// TIA Portal V19 export
FUNCTION_BLOCK "A01_HMI_FB"   // FB75, LAD
TITLE = HMI Managment
AUTHOR : Piemme
FAMILY : System
// stored: MemoryReserve 100, SetENOAutomatically false
   VAR
      MB1_Decoder { ExternalAccessible := 'False'; ExternalVisible := 'False'; ExternalWritable := 'False'} : "ButtonsHMIDecoder";
   END_VAR
   VAR CONSTANT
      "1001_HU_AREA01" : Int := 1001;
      "1002_HU_DECOILER" : Int := 1002;
      "1011_DECOILER_IN_LINE_FEED" : Int := 1011;
      "1012_DECOILER_IN_LINE_JAWS" : Int := 1012;
      "1013_DECOILER_IN_LINE_COUPLING" : Int := 1013;
      "1014_DECOILER_IN_LINE_SNUBBER_LIFT" : Int := 1014;
      "1015_DECOILER_IN_LINE_SNUBBER_ROL" : Int := 1015;
      "1016_DECOILER_IN_LINE_BRAKE_OPEN" : Int := 1016;
      "1017_DECOILER_IN_LINE_BRAKE_PARTIAL" : Int := 1017;
      "1021_DECOILER_OUT_LINE_FEED" : Int := 1021;
      "1022_DECOILER_OUT_LINE_JAWS" : Int := 1022;
      "1023_DECOILER_OUT_LINE_COUPLING" : Int := 1023;
      "1024_DECOILER_OUT_LINE_SNUBBER_LIFT" : Int := 1024;
      "1025_DECOILER_OUT_LINE_SNUBBER_ROL" : Int := 1025;
      "1026_DECOILER_OUT_LINE_BRAKE_OPEN" : Int := 1026;
      "1027_DECOILER_OUT_LINE_BRAKE_PARTIAL" : Int := 1027;
      "1031_DECOILER_ROTATION" : Int := 1031;
      "1032_DECOILER_ROTATION_DIR" : Int := 1032;
      "1033_DECOILER_ROTATION_PIVOT" : Int := 1033;
      "1034_DECOILER_TRASLATION_BWD_FWD" : Int := 1034;
      "1035_DECOILER_TRANSLATION_MOVE_TO_POS" : Int := 1035;
      "1041_PEELER_LIFT" : Int := 1041;
      "1042_PEELER_EXTENSION" : Int := 1042;
      "1051_STRAIGHTENER_MOVE" : Int := 1051;
      "1052_STRAIGHTENER_LIFT_ENTRYROLL" : Int := 1052;
      "1053_STRAIGHTENER_LIFT_EXITROLL" : Int := 1053;
      "1054_STRAIGHTENER_COUPLING" : Int := 1054;
      "1061_JB_CUT" : Int := 1061;
      "1062_JB_TORCH_MOVE" : Int := 1062;
      "1063_JB_ENTRYCLAMP" : Int := 1063;
      "1064_JB_EXITCLAMP" : Int := 1064;
      "1065_JB_WELDER" : Int := 1065;
      "1066_JB_WELD_CYCLE" : Int := 1066;
      "1071_JB_PINCHROLL_MOVE" : Int := 1071;
      "1072_JB_PINCHROLL_LIFT" : Int := 1072;
      "1073_JB_PINCHROLL_COUPLING" : Int := 1073;
      "1081_LOOP1" : Int := 1081;
   END_VAR
   VAR_TEMP   // added for the SCL form of the ladder/FBD networks
      _w1 : Bool;
      _w2 : Bool;
   END_VAR
BEGIN

REGION Network 2: <<< MB1 MANUALS OPERATIONS >>>
END_REGION

REGION Network 3 (SCL): Reset Op
   #MB1_Decoder.OpEnabled := FALSE;
   #MB1_Decoder.OpRunning := FALSE;
   #MB1_Decoder.OpDone := FALSE;
END_REGION

REGION Network 4: MB1 Code 1001 - Area 01 HU
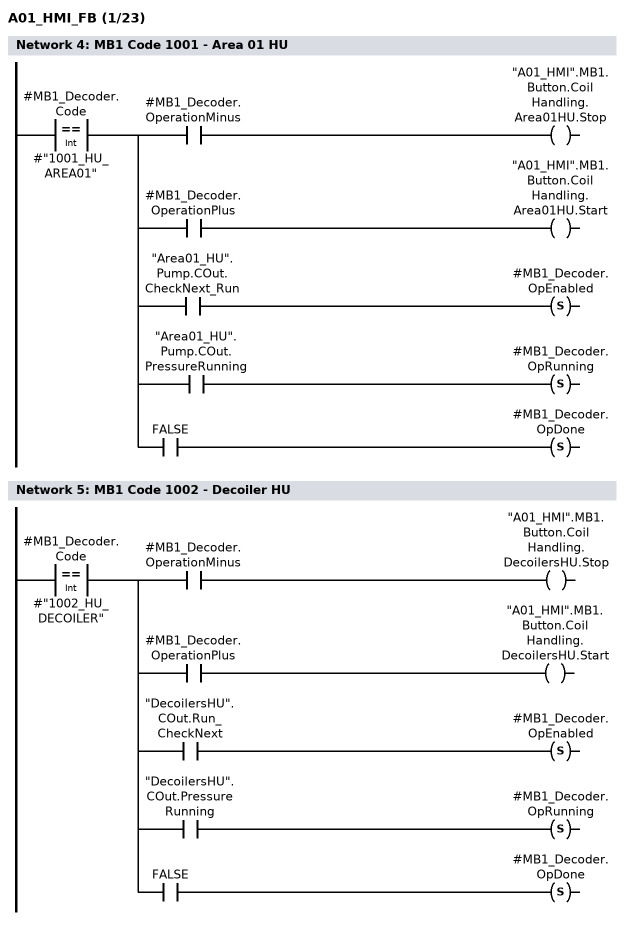
   RUNG wire#powerrail
      { S7_Templates := "SrcType := Int" } EQ_Contact(in1 := #MB1_Decoder.Code, in2 := #"1001_HU_AREA01")
      wire#w1
      Contact( #MB1_Decoder.OperationMinus )
      Coil( "A01_HMI".MB1.Button.CoilHandling.Area01HU.Stop )
   END_RUNG
   RUNG wire#w1
      Contact( #MB1_Decoder.OperationPlus )
      Coil( "A01_HMI".MB1.Button.CoilHandling.Area01HU.Start )
   END_RUNG
   RUNG wire#w1
      Contact( "Area01_HU".Pump.COut.CheckNext_Run )
      S_Coil( #MB1_Decoder.OpEnabled )
   END_RUNG
   RUNG wire#w1
      Contact( "Area01_HU".Pump.COut.PressureRunning )
      S_Coil( #MB1_Decoder.OpRunning )
   END_RUNG
   RUNG wire#w1
      Contact( FALSE )
      S_Coil( #MB1_Decoder.OpDone )
   END_RUNG
   // the same network as SCL:
   #_w1 := #MB1_Decoder.Code = #"1001_HU_AREA01";
   "A01_HMI".MB1.Button.CoilHandling.Area01HU.Stop := #_w1 AND #MB1_Decoder.OperationMinus;
   "A01_HMI".MB1.Button.CoilHandling.Area01HU.Start := #_w1 AND #MB1_Decoder.OperationPlus;
   IF #_w1 AND "Area01_HU".Pump.COut.CheckNext_Run THEN #MB1_Decoder.OpEnabled := TRUE; END_IF;
   IF #_w1 AND "Area01_HU".Pump.COut.PressureRunning THEN #MB1_Decoder.OpRunning := TRUE; END_IF;
   IF #_w1 AND FALSE THEN #MB1_Decoder.OpDone := TRUE; END_IF;
END_REGION

REGION Network 5: MB1 Code 1002 - Decoiler HU
   RUNG wire#powerrail
      { S7_Templates := "SrcType := Int" } EQ_Contact(in1 := #MB1_Decoder.Code, in2 := #"1002_HU_DECOILER")
      wire#w1
      Contact( #MB1_Decoder.OperationMinus )
      Coil( "A01_HMI".MB1.Button.CoilHandling.DecoilersHU.Stop )
   END_RUNG
   RUNG wire#w1
      Contact( #MB1_Decoder.OperationPlus )
      Coil( "A01_HMI".MB1.Button.CoilHandling.DecoilersHU.Start )
   END_RUNG
   RUNG wire#w1
      Contact( "DecoilersHU".COut.Run_CheckNext )
      S_Coil( #MB1_Decoder.OpEnabled )
   END_RUNG
   RUNG wire#w1
      Contact( "DecoilersHU".COut.PressureRunning )
      S_Coil( #MB1_Decoder.OpRunning )
   END_RUNG
   RUNG wire#w1
      Contact( FALSE )
      S_Coil( #MB1_Decoder.OpDone )
   END_RUNG
   // the same network as SCL:
   #_w1 := #MB1_Decoder.Code = #"1002_HU_DECOILER";
   "A01_HMI".MB1.Button.CoilHandling.DecoilersHU.Stop := #_w1 AND #MB1_Decoder.OperationMinus;
   "A01_HMI".MB1.Button.CoilHandling.DecoilersHU.Start := #_w1 AND #MB1_Decoder.OperationPlus;
   IF #_w1 AND "DecoilersHU".COut.Run_CheckNext THEN #MB1_Decoder.OpEnabled := TRUE; END_IF;
   IF #_w1 AND "DecoilersHU".COut.PressureRunning THEN #MB1_Decoder.OpRunning := TRUE; END_IF;
   IF #_w1 AND FALSE THEN #MB1_Decoder.OpDone := TRUE; END_IF;
END_REGION

REGION Network 6: MB1 Code 1011 - Decoiler In Line bkw / fwd
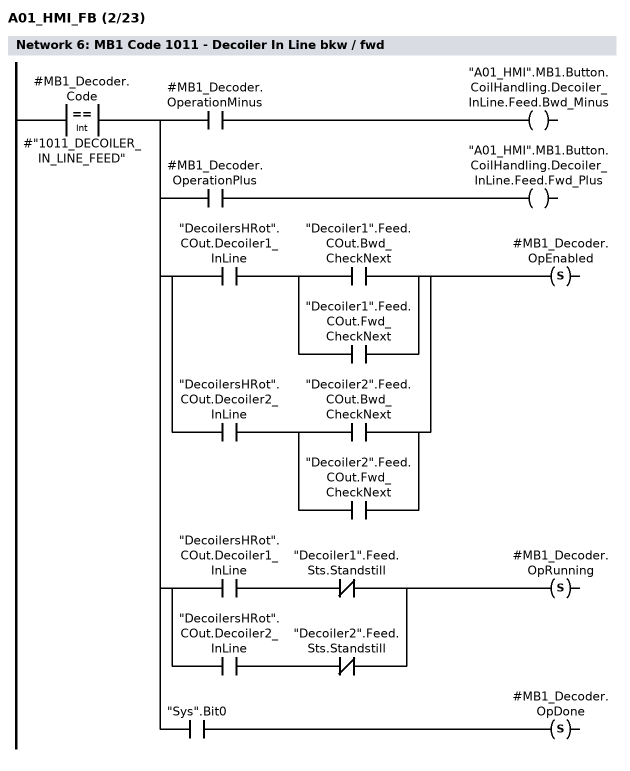
   RUNG wire#powerrail
      { S7_Templates := "SrcType := Int" } EQ_Contact(in1 := #MB1_Decoder.Code, in2 := #"1011_DECOILER_IN_LINE_FEED")
      wire#w1
      Contact( #MB1_Decoder.OperationMinus )
      Coil( "A01_HMI".MB1.Button.CoilHandling.Decoiler_InLine.Feed.Bwd_Minus )
   END_RUNG
   RUNG wire#w1
      Contact( #MB1_Decoder.OperationPlus )
      Coil( "A01_HMI".MB1.Button.CoilHandling.Decoiler_InLine.Feed.Fwd_Plus )
   END_RUNG
   RUNG wire#w1
      Contact( "DecoilersHRot".COut.Decoiler1_InLine )
      wire#w2
      Contact( "Decoiler1".Feed.COut.Bwd_CheckNext )
      wire#w3
      S_Coil( #MB1_Decoder.OpEnabled )
   END_RUNG
   RUNG wire#w2
      Contact( "Decoiler1".Feed.COut.Fwd_CheckNext )
   END_RUNG wire#w3
   RUNG wire#w1
      Contact( "DecoilersHRot".COut.Decoiler2_InLine )
      wire#w4
      Contact( "Decoiler2".Feed.COut.Bwd_CheckNext )
   END_RUNG wire#w3
   RUNG wire#w4
      Contact( "Decoiler2".Feed.COut.Fwd_CheckNext )
   END_RUNG wire#w3
   RUNG wire#w1
      Contact( "DecoilersHRot".COut.Decoiler1_InLine )
      I_Contact( "Decoiler1".Feed.Sts.Standstill )
      wire#w5
      S_Coil( #MB1_Decoder.OpRunning )
   END_RUNG
   RUNG wire#w1
      Contact( "DecoilersHRot".COut.Decoiler2_InLine )
      I_Contact( "Decoiler2".Feed.Sts.Standstill )
   END_RUNG wire#w5
   RUNG wire#w1
      Contact( "Sys".Bit0 )
      S_Coil( #MB1_Decoder.OpDone )
   END_RUNG
   // the same network as SCL:
   #_w1 := #MB1_Decoder.Code = #"1011_DECOILER_IN_LINE_FEED";
   "A01_HMI".MB1.Button.CoilHandling.Decoiler_InLine.Feed.Bwd_Minus := #_w1 AND #MB1_Decoder.OperationMinus;
   "A01_HMI".MB1.Button.CoilHandling.Decoiler_InLine.Feed.Fwd_Plus := #_w1 AND #MB1_Decoder.OperationPlus;
   IF #_w1 AND (("DecoilersHRot".COut.Decoiler1_InLine AND ("Decoiler1".Feed.COut.Bwd_CheckNext OR "Decoiler1".Feed.COut.Fwd_CheckNext)) OR ("DecoilersHRot".COut.Decoiler2_InLine AND ("Decoiler2".Feed.COut.Bwd_CheckNext OR "Decoiler2".Feed.COut.Fwd_CheckNext))) THEN
       #MB1_Decoder.OpEnabled := TRUE;
   END_IF;
   IF #_w1 AND (("DecoilersHRot".COut.Decoiler1_InLine AND NOT "Decoiler1".Feed.Sts.Standstill) OR ("DecoilersHRot".COut.Decoiler2_InLine AND NOT "Decoiler2".Feed.Sts.Standstill)) THEN
       #MB1_Decoder.OpRunning := TRUE;
   END_IF;
   IF #_w1 AND "Sys".Bit0 THEN #MB1_Decoder.OpDone := TRUE; END_IF;
END_REGION

REGION Network 7: MB1 Code 1012 - Decoiler In Line jaws open / close
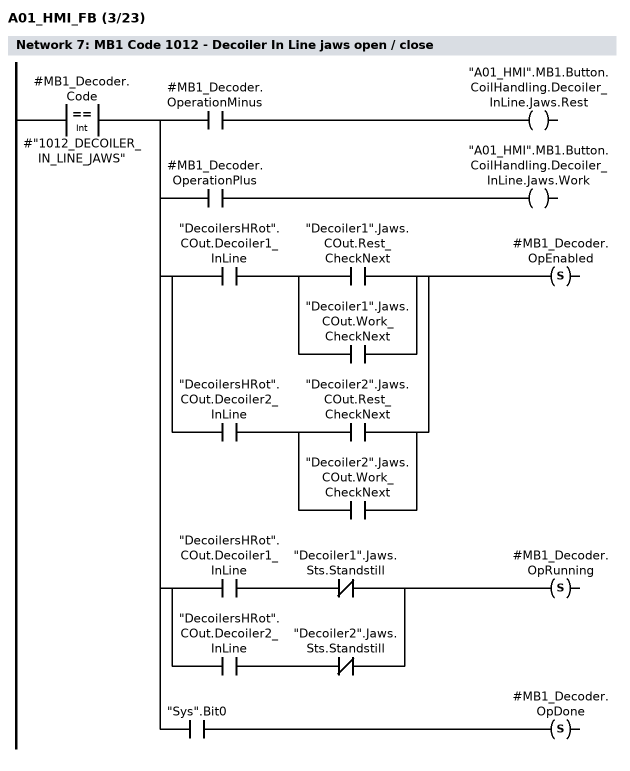
   RUNG wire#powerrail
      { S7_Templates := "SrcType := Int" } EQ_Contact(in1 := #MB1_Decoder.Code, in2 := #"1012_DECOILER_IN_LINE_JAWS")
      wire#w1
      Contact( #MB1_Decoder.OperationMinus )
      Coil( "A01_HMI".MB1.Button.CoilHandling.Decoiler_InLine.Jaws.Rest )
   END_RUNG
   RUNG wire#w1
      Contact( #MB1_Decoder.OperationPlus )
      Coil( "A01_HMI".MB1.Button.CoilHandling.Decoiler_InLine.Jaws.Work )
   END_RUNG
   RUNG wire#w1
      Contact( "DecoilersHRot".COut.Decoiler1_InLine )
      wire#w2
      Contact( "Decoiler1".Jaws.COut.Rest_CheckNext )
      wire#w3
      S_Coil( #MB1_Decoder.OpEnabled )
   END_RUNG
   RUNG wire#w2
      Contact( "Decoiler1".Jaws.COut.Work_CheckNext )
   END_RUNG wire#w3
   RUNG wire#w1
      Contact( "DecoilersHRot".COut.Decoiler2_InLine )
      wire#w4
      Contact( "Decoiler2".Jaws.COut.Rest_CheckNext )
   END_RUNG wire#w3
   RUNG wire#w4
      Contact( "Decoiler2".Jaws.COut.Work_CheckNext )
   END_RUNG wire#w3
   RUNG wire#w1
      Contact( "DecoilersHRot".COut.Decoiler1_InLine )
      I_Contact( "Decoiler1".Jaws.Sts.Standstill )
      wire#w5
      S_Coil( #MB1_Decoder.OpRunning )
   END_RUNG
   RUNG wire#w1
      Contact( "DecoilersHRot".COut.Decoiler2_InLine )
      I_Contact( "Decoiler2".Jaws.Sts.Standstill )
   END_RUNG wire#w5
   RUNG wire#w1
      Contact( "Sys".Bit0 )
      S_Coil( #MB1_Decoder.OpDone )
   END_RUNG
   // the same network as SCL:
   #_w1 := #MB1_Decoder.Code = #"1012_DECOILER_IN_LINE_JAWS";
   "A01_HMI".MB1.Button.CoilHandling.Decoiler_InLine.Jaws.Rest := #_w1 AND #MB1_Decoder.OperationMinus;
   "A01_HMI".MB1.Button.CoilHandling.Decoiler_InLine.Jaws.Work := #_w1 AND #MB1_Decoder.OperationPlus;
   IF #_w1 AND (("DecoilersHRot".COut.Decoiler1_InLine AND ("Decoiler1".Jaws.COut.Rest_CheckNext OR "Decoiler1".Jaws.COut.Work_CheckNext)) OR ("DecoilersHRot".COut.Decoiler2_InLine AND ("Decoiler2".Jaws.COut.Rest_CheckNext OR "Decoiler2".Jaws.COut.Work_CheckNext))) THEN
       #MB1_Decoder.OpEnabled := TRUE;
   END_IF;
   IF #_w1 AND (("DecoilersHRot".COut.Decoiler1_InLine AND NOT "Decoiler1".Jaws.Sts.Standstill) OR ("DecoilersHRot".COut.Decoiler2_InLine AND NOT "Decoiler2".Jaws.Sts.Standstill)) THEN
       #MB1_Decoder.OpRunning := TRUE;
   END_IF;
   IF #_w1 AND "Sys".Bit0 THEN #MB1_Decoder.OpDone := TRUE; END_IF;
END_REGION

REGION Network 8: MB1 Code 1013 - Decoiler In Line motor coupling rest / work
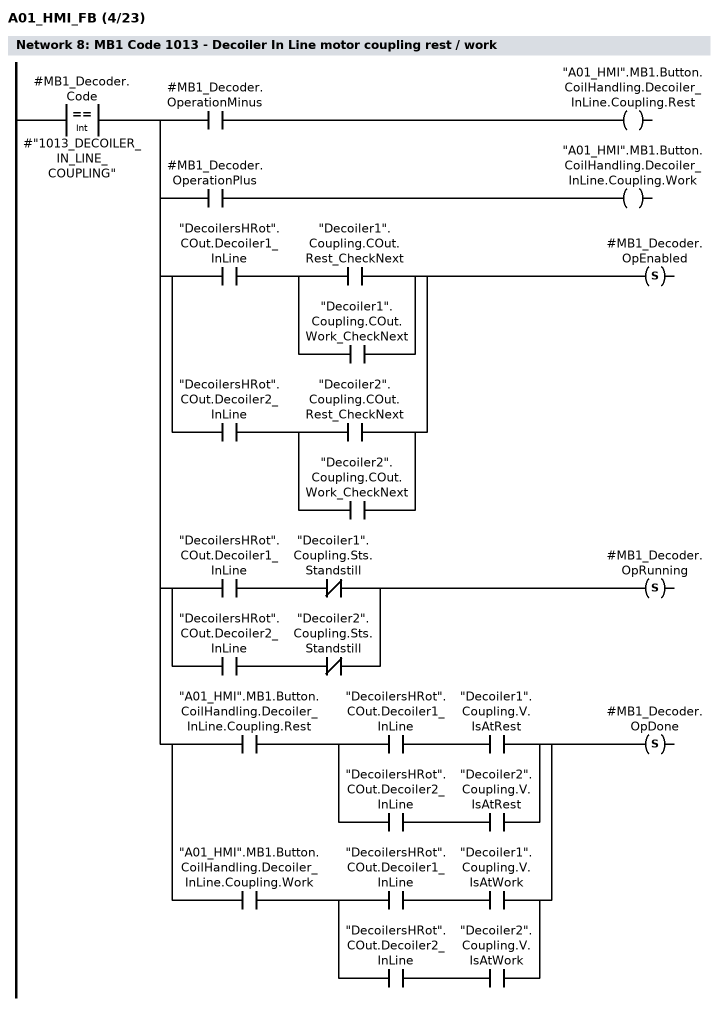
   RUNG wire#powerrail
      { S7_Templates := "SrcType := Int" } EQ_Contact(in1 := #MB1_Decoder.Code, in2 := #"1013_DECOILER_IN_LINE_COUPLING")
      wire#w1
      Contact( #MB1_Decoder.OperationMinus )
      Coil( "A01_HMI".MB1.Button.CoilHandling.Decoiler_InLine.Coupling.Rest )
   END_RUNG
   RUNG wire#w1
      Contact( #MB1_Decoder.OperationPlus )
      Coil( "A01_HMI".MB1.Button.CoilHandling.Decoiler_InLine.Coupling.Work )
   END_RUNG
   RUNG wire#w1
      Contact( "DecoilersHRot".COut.Decoiler1_InLine )
      wire#w2
      Contact( "Decoiler1".Coupling.COut.Rest_CheckNext )
      wire#w3
      S_Coil( #MB1_Decoder.OpEnabled )
   END_RUNG
   RUNG wire#w2
      Contact( "Decoiler1".Coupling.COut.Work_CheckNext )
   END_RUNG wire#w3
   RUNG wire#w1
      Contact( "DecoilersHRot".COut.Decoiler2_InLine )
      wire#w4
      Contact( "Decoiler2".Coupling.COut.Rest_CheckNext )
   END_RUNG wire#w3
   RUNG wire#w4
      Contact( "Decoiler2".Coupling.COut.Work_CheckNext )
   END_RUNG wire#w3
   RUNG wire#w1
      Contact( "DecoilersHRot".COut.Decoiler1_InLine )
      I_Contact( "Decoiler1".Coupling.Sts.Standstill )
      wire#w5
      S_Coil( #MB1_Decoder.OpRunning )
   END_RUNG
   RUNG wire#w1
      Contact( "DecoilersHRot".COut.Decoiler2_InLine )
      I_Contact( "Decoiler2".Coupling.Sts.Standstill )
   END_RUNG wire#w5
   RUNG wire#w1
      Contact( "A01_HMI".MB1.Button.CoilHandling.Decoiler_InLine.Coupling.Rest )
      wire#w6
      Contact( "DecoilersHRot".COut.Decoiler1_InLine )
      Contact( "Decoiler1".Coupling.V.IsAtRest )
      wire#w7
      S_Coil( #MB1_Decoder.OpDone )
   END_RUNG
   RUNG wire#w6
      Contact( "DecoilersHRot".COut.Decoiler2_InLine )
      Contact( "Decoiler2".Coupling.V.IsAtRest )
   END_RUNG wire#w7
   RUNG wire#w1
      Contact( "A01_HMI".MB1.Button.CoilHandling.Decoiler_InLine.Coupling.Work )
      wire#w8
      Contact( "DecoilersHRot".COut.Decoiler1_InLine )
      Contact( "Decoiler1".Coupling.V.IsAtWork )
   END_RUNG wire#w7
   RUNG wire#w8
      Contact( "DecoilersHRot".COut.Decoiler2_InLine )
      Contact( "Decoiler2".Coupling.V.IsAtWork )
   END_RUNG wire#w7
   // the same network as SCL:
   #_w1 := #MB1_Decoder.Code = #"1013_DECOILER_IN_LINE_COUPLING";
   "A01_HMI".MB1.Button.CoilHandling.Decoiler_InLine.Coupling.Rest := #_w1 AND #MB1_Decoder.OperationMinus;
   "A01_HMI".MB1.Button.CoilHandling.Decoiler_InLine.Coupling.Work := #_w1 AND #MB1_Decoder.OperationPlus;
   IF #_w1 AND (("DecoilersHRot".COut.Decoiler1_InLine AND ("Decoiler1".Coupling.COut.Rest_CheckNext OR "Decoiler1".Coupling.COut.Work_CheckNext)) OR ("DecoilersHRot".COut.Decoiler2_InLine AND ("Decoiler2".Coupling.COut.Rest_CheckNext OR "Decoiler2".Coupling.COut.Work_CheckNext))) THEN
       #MB1_Decoder.OpEnabled := TRUE;
   END_IF;
   IF #_w1 AND (("DecoilersHRot".COut.Decoiler1_InLine AND NOT "Decoiler1".Coupling.Sts.Standstill) OR ("DecoilersHRot".COut.Decoiler2_InLine AND NOT "Decoiler2".Coupling.Sts.Standstill)) THEN
       #MB1_Decoder.OpRunning := TRUE;
   END_IF;
   IF #_w1 AND (("A01_HMI".MB1.Button.CoilHandling.Decoiler_InLine.Coupling.Rest AND (("DecoilersHRot".COut.Decoiler1_InLine AND "Decoiler1".Coupling.V.IsAtRest) OR ("DecoilersHRot".COut.Decoiler2_InLine AND "Decoiler2".Coupling.V.IsAtRest))) OR ("A01_HMI".MB1.Button.CoilHandling.Decoiler_InLine.Coupling.Work AND (("DecoilersHRot".COut.Decoiler1_InLine AND "Decoiler1".Coupling.V.IsAtWork) OR ("DecoilersHRot".COut.Decoiler2_InLine AND "Decoiler2".Coupling.V.IsAtWork)))) THEN
       #MB1_Decoder.OpDone := TRUE;
   END_IF;
END_REGION

REGION Network 9: MB1 Code 1014 - Decoiler In Line snubber lift up / down
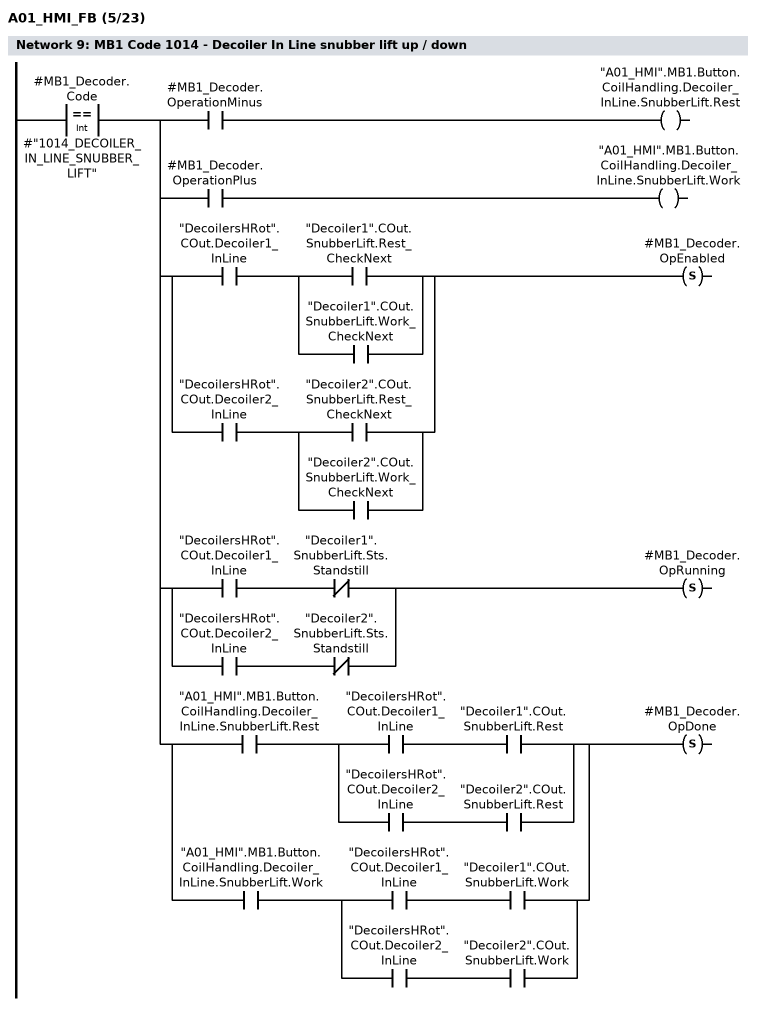
   RUNG wire#powerrail
      { S7_Templates := "SrcType := Int" } EQ_Contact(in1 := #MB1_Decoder.Code, in2 := #"1014_DECOILER_IN_LINE_SNUBBER_LIFT")
      wire#w1
      Contact( #MB1_Decoder.OperationMinus )
      Coil( "A01_HMI".MB1.Button.CoilHandling.Decoiler_InLine.SnubberLift.Rest )
   END_RUNG
   RUNG wire#w1
      Contact( #MB1_Decoder.OperationPlus )
      Coil( "A01_HMI".MB1.Button.CoilHandling.Decoiler_InLine.SnubberLift.Work )
   END_RUNG
   RUNG wire#w1
      Contact( "DecoilersHRot".COut.Decoiler1_InLine )
      wire#w2
      Contact( "Decoiler1".COut.SnubberLift.Rest_CheckNext )
      wire#w3
      S_Coil( #MB1_Decoder.OpEnabled )
   END_RUNG
   RUNG wire#w2
      Contact( "Decoiler1".COut.SnubberLift.Work_CheckNext )
   END_RUNG wire#w3
   RUNG wire#w1
      Contact( "DecoilersHRot".COut.Decoiler2_InLine )
      wire#w4
      Contact( "Decoiler2".COut.SnubberLift.Rest_CheckNext )
   END_RUNG wire#w3
   RUNG wire#w4
      Contact( "Decoiler2".COut.SnubberLift.Work_CheckNext )
   END_RUNG wire#w3
   RUNG wire#w1
      Contact( "DecoilersHRot".COut.Decoiler1_InLine )
      I_Contact( "Decoiler1".SnubberLift.Sts.Standstill )
      wire#w5
      S_Coil( #MB1_Decoder.OpRunning )
   END_RUNG
   RUNG wire#w1
      Contact( "DecoilersHRot".COut.Decoiler2_InLine )
      I_Contact( "Decoiler2".SnubberLift.Sts.Standstill )
   END_RUNG wire#w5
   RUNG wire#w1
      Contact( "A01_HMI".MB1.Button.CoilHandling.Decoiler_InLine.SnubberLift.Rest )
      wire#w6
      Contact( "DecoilersHRot".COut.Decoiler1_InLine )
      Contact( "Decoiler1".COut.SnubberLift.Rest )
      wire#w7
      S_Coil( #MB1_Decoder.OpDone )
   END_RUNG
   RUNG wire#w6
      Contact( "DecoilersHRot".COut.Decoiler2_InLine )
      Contact( "Decoiler2".COut.SnubberLift.Rest )
   END_RUNG wire#w7
   RUNG wire#w1
      Contact( "A01_HMI".MB1.Button.CoilHandling.Decoiler_InLine.SnubberLift.Work )
      wire#w8
      Contact( "DecoilersHRot".COut.Decoiler1_InLine )
      Contact( "Decoiler1".COut.SnubberLift.Work )
   END_RUNG wire#w7
   RUNG wire#w8
      Contact( "DecoilersHRot".COut.Decoiler2_InLine )
      Contact( "Decoiler2".COut.SnubberLift.Work )
   END_RUNG wire#w7
   // the same network as SCL:
   #_w1 := #MB1_Decoder.Code = #"1014_DECOILER_IN_LINE_SNUBBER_LIFT";
   "A01_HMI".MB1.Button.CoilHandling.Decoiler_InLine.SnubberLift.Rest := #_w1 AND #MB1_Decoder.OperationMinus;
   "A01_HMI".MB1.Button.CoilHandling.Decoiler_InLine.SnubberLift.Work := #_w1 AND #MB1_Decoder.OperationPlus;
   IF #_w1 AND (("DecoilersHRot".COut.Decoiler1_InLine AND ("Decoiler1".COut.SnubberLift.Rest_CheckNext OR "Decoiler1".COut.SnubberLift.Work_CheckNext)) OR ("DecoilersHRot".COut.Decoiler2_InLine AND ("Decoiler2".COut.SnubberLift.Rest_CheckNext OR "Decoiler2".COut.SnubberLift.Work_CheckNext))) THEN
       #MB1_Decoder.OpEnabled := TRUE;
   END_IF;
   IF #_w1 AND (("DecoilersHRot".COut.Decoiler1_InLine AND NOT "Decoiler1".SnubberLift.Sts.Standstill) OR ("DecoilersHRot".COut.Decoiler2_InLine AND NOT "Decoiler2".SnubberLift.Sts.Standstill)) THEN
       #MB1_Decoder.OpRunning := TRUE;
   END_IF;
   IF #_w1 AND (("A01_HMI".MB1.Button.CoilHandling.Decoiler_InLine.SnubberLift.Rest AND (("DecoilersHRot".COut.Decoiler1_InLine AND "Decoiler1".COut.SnubberLift.Rest) OR ("DecoilersHRot".COut.Decoiler2_InLine AND "Decoiler2".COut.SnubberLift.Rest))) OR ("A01_HMI".MB1.Button.CoilHandling.Decoiler_InLine.SnubberLift.Work AND (("DecoilersHRot".COut.Decoiler1_InLine AND "Decoiler1".COut.SnubberLift.Work) OR ("DecoilersHRot".COut.Decoiler2_InLine AND "Decoiler2".COut.SnubberLift.Work)))) THEN
       #MB1_Decoder.OpDone := TRUE;
   END_IF;
END_REGION

REGION Network 10: MB1 Code 1015 - Decoiler In Line nubber roll bkw / fwd
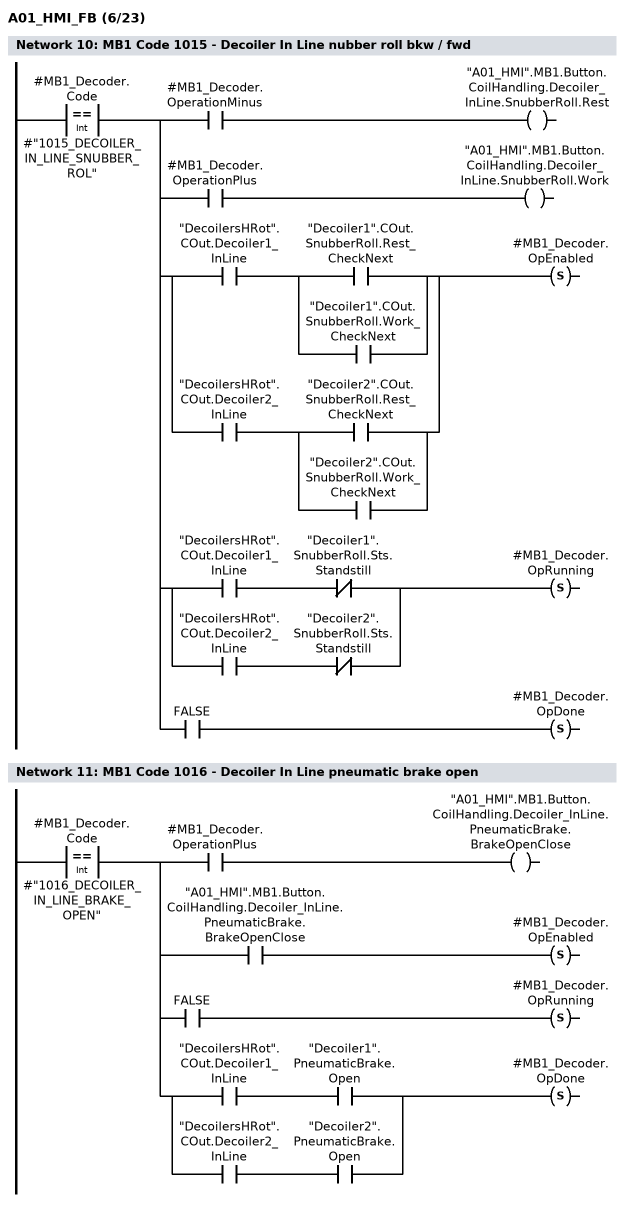
   RUNG wire#powerrail
      { S7_Templates := "SrcType := Int" } EQ_Contact(in1 := #MB1_Decoder.Code, in2 := #"1015_DECOILER_IN_LINE_SNUBBER_ROL")
      wire#w1
      Contact( #MB1_Decoder.OperationMinus )
      Coil( "A01_HMI".MB1.Button.CoilHandling.Decoiler_InLine.SnubberRoll.Rest )
   END_RUNG
   RUNG wire#w1
      Contact( #MB1_Decoder.OperationPlus )
      Coil( "A01_HMI".MB1.Button.CoilHandling.Decoiler_InLine.SnubberRoll.Work )
   END_RUNG
   RUNG wire#w1
      Contact( "DecoilersHRot".COut.Decoiler1_InLine )
      wire#w2
      Contact( "Decoiler1".COut.SnubberRoll.Rest_CheckNext )
      wire#w3
      S_Coil( #MB1_Decoder.OpEnabled )
   END_RUNG
   RUNG wire#w2
      Contact( "Decoiler1".COut.SnubberRoll.Work_CheckNext )
   END_RUNG wire#w3
   RUNG wire#w1
      Contact( "DecoilersHRot".COut.Decoiler2_InLine )
      wire#w4
      Contact( "Decoiler2".COut.SnubberRoll.Rest_CheckNext )
   END_RUNG wire#w3
   RUNG wire#w4
      Contact( "Decoiler2".COut.SnubberRoll.Work_CheckNext )
   END_RUNG wire#w3
   RUNG wire#w1
      Contact( "DecoilersHRot".COut.Decoiler1_InLine )
      I_Contact( "Decoiler1".SnubberRoll.Sts.Standstill )
      wire#w5
      S_Coil( #MB1_Decoder.OpRunning )
   END_RUNG
   RUNG wire#w1
      Contact( "DecoilersHRot".COut.Decoiler2_InLine )
      I_Contact( "Decoiler2".SnubberRoll.Sts.Standstill )
   END_RUNG wire#w5
   RUNG wire#w1
      Contact( FALSE )
      S_Coil( #MB1_Decoder.OpDone )
   END_RUNG
   // the same network as SCL:
   #_w1 := #MB1_Decoder.Code = #"1015_DECOILER_IN_LINE_SNUBBER_ROL";
   "A01_HMI".MB1.Button.CoilHandling.Decoiler_InLine.SnubberRoll.Rest := #_w1 AND #MB1_Decoder.OperationMinus;
   "A01_HMI".MB1.Button.CoilHandling.Decoiler_InLine.SnubberRoll.Work := #_w1 AND #MB1_Decoder.OperationPlus;
   IF #_w1 AND (("DecoilersHRot".COut.Decoiler1_InLine AND ("Decoiler1".COut.SnubberRoll.Rest_CheckNext OR "Decoiler1".COut.SnubberRoll.Work_CheckNext)) OR ("DecoilersHRot".COut.Decoiler2_InLine AND ("Decoiler2".COut.SnubberRoll.Rest_CheckNext OR "Decoiler2".COut.SnubberRoll.Work_CheckNext))) THEN
       #MB1_Decoder.OpEnabled := TRUE;
   END_IF;
   IF #_w1 AND (("DecoilersHRot".COut.Decoiler1_InLine AND NOT "Decoiler1".SnubberRoll.Sts.Standstill) OR ("DecoilersHRot".COut.Decoiler2_InLine AND NOT "Decoiler2".SnubberRoll.Sts.Standstill)) THEN
       #MB1_Decoder.OpRunning := TRUE;
   END_IF;
   IF #_w1 AND FALSE THEN #MB1_Decoder.OpDone := TRUE; END_IF;
END_REGION

REGION Network 11: MB1 Code 1016 - Decoiler In Line pneumatic brake open
   RUNG wire#powerrail
      { S7_Templates := "SrcType := Int" } EQ_Contact(in1 := #MB1_Decoder.Code, in2 := #"1016_DECOILER_IN_LINE_BRAKE_OPEN")
      wire#w1
      Contact( #MB1_Decoder.OperationPlus )
      Coil( "A01_HMI".MB1.Button.CoilHandling.Decoiler_InLine.PneumaticBrake.BrakeOpenClose )
   END_RUNG
   RUNG wire#w1
      Contact( "A01_HMI".MB1.Button.CoilHandling.Decoiler_InLine.PneumaticBrake.BrakeOpenClose )
      S_Coil( #MB1_Decoder.OpEnabled )
   END_RUNG
   RUNG wire#w1
      Contact( FALSE )
      S_Coil( #MB1_Decoder.OpRunning )
   END_RUNG
   RUNG wire#w1
      Contact( "DecoilersHRot".COut.Decoiler1_InLine )
      Contact( "Decoiler1".PneumaticBrake.Open )
      wire#w2
      S_Coil( #MB1_Decoder.OpDone )
   END_RUNG
   RUNG wire#w1
      Contact( "DecoilersHRot".COut.Decoiler2_InLine )
      Contact( "Decoiler2".PneumaticBrake.Open )
   END_RUNG wire#w2
   // the same network as SCL:
   #_w1 := #MB1_Decoder.Code = #"1016_DECOILER_IN_LINE_BRAKE_OPEN";
   "A01_HMI".MB1.Button.CoilHandling.Decoiler_InLine.PneumaticBrake.BrakeOpenClose := #_w1 AND #MB1_Decoder.OperationPlus;
   IF #_w1 AND "A01_HMI".MB1.Button.CoilHandling.Decoiler_InLine.PneumaticBrake.BrakeOpenClose THEN
       #MB1_Decoder.OpEnabled := TRUE;
   END_IF;
   IF #_w1 AND FALSE THEN #MB1_Decoder.OpRunning := TRUE; END_IF;
   IF #_w1 AND (("DecoilersHRot".COut.Decoiler1_InLine AND "Decoiler1".PneumaticBrake.Open) OR ("DecoilersHRot".COut.Decoiler2_InLine AND "Decoiler2".PneumaticBrake.Open)) THEN
       #MB1_Decoder.OpDone := TRUE;
   END_IF;
END_REGION

REGION Network 12: MB1 Code 1017 - Decoiler In Line pneumatic brake partial
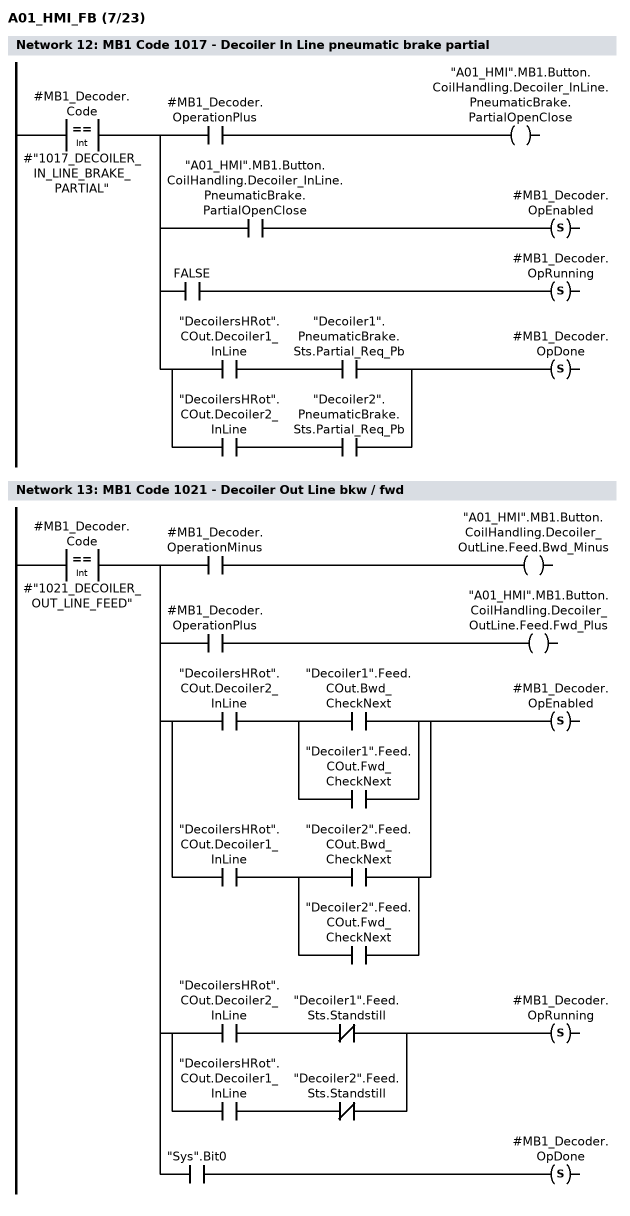
   RUNG wire#powerrail
      { S7_Templates := "SrcType := Int" } EQ_Contact(in1 := #MB1_Decoder.Code, in2 := #"1017_DECOILER_IN_LINE_BRAKE_PARTIAL")
      wire#w1
      Contact( #MB1_Decoder.OperationPlus )
      Coil( "A01_HMI".MB1.Button.CoilHandling.Decoiler_InLine.PneumaticBrake.PartialOpenClose )
   END_RUNG
   RUNG wire#w1
      Contact( "A01_HMI".MB1.Button.CoilHandling.Decoiler_InLine.PneumaticBrake.PartialOpenClose )
      S_Coil( #MB1_Decoder.OpEnabled )
   END_RUNG
   RUNG wire#w1
      Contact( FALSE )
      S_Coil( #MB1_Decoder.OpRunning )
   END_RUNG
   RUNG wire#w1
      Contact( "DecoilersHRot".COut.Decoiler1_InLine )
      Contact( "Decoiler1".PneumaticBrake.Sts.Partial_Req_Pb )
      wire#w2
      S_Coil( #MB1_Decoder.OpDone )
   END_RUNG
   RUNG wire#w1
      Contact( "DecoilersHRot".COut.Decoiler2_InLine )
      Contact( "Decoiler2".PneumaticBrake.Sts.Partial_Req_Pb )
   END_RUNG wire#w2
   // the same network as SCL:
   #_w1 := #MB1_Decoder.Code = #"1017_DECOILER_IN_LINE_BRAKE_PARTIAL";
   "A01_HMI".MB1.Button.CoilHandling.Decoiler_InLine.PneumaticBrake.PartialOpenClose := #_w1 AND #MB1_Decoder.OperationPlus;
   IF #_w1 AND "A01_HMI".MB1.Button.CoilHandling.Decoiler_InLine.PneumaticBrake.PartialOpenClose THEN
       #MB1_Decoder.OpEnabled := TRUE;
   END_IF;
   IF #_w1 AND FALSE THEN #MB1_Decoder.OpRunning := TRUE; END_IF;
   IF #_w1 AND (("DecoilersHRot".COut.Decoiler1_InLine AND "Decoiler1".PneumaticBrake.Sts.Partial_Req_Pb) OR ("DecoilersHRot".COut.Decoiler2_InLine AND "Decoiler2".PneumaticBrake.Sts.Partial_Req_Pb)) THEN
       #MB1_Decoder.OpDone := TRUE;
   END_IF;
END_REGION

REGION Network 13: MB1 Code 1021 - Decoiler Out Line bkw / fwd
   RUNG wire#powerrail
      { S7_Templates := "SrcType := Int" } EQ_Contact(in1 := #MB1_Decoder.Code, in2 := #"1021_DECOILER_OUT_LINE_FEED")
      wire#w1
      Contact( #MB1_Decoder.OperationMinus )
      Coil( "A01_HMI".MB1.Button.CoilHandling.Decoiler_OutLine.Feed.Bwd_Minus )
   END_RUNG
   RUNG wire#w1
      Contact( #MB1_Decoder.OperationPlus )
      Coil( "A01_HMI".MB1.Button.CoilHandling.Decoiler_OutLine.Feed.Fwd_Plus )
   END_RUNG
   RUNG wire#w1
      Contact( "DecoilersHRot".COut.Decoiler2_InLine )
      wire#w2
      Contact( "Decoiler1".Feed.COut.Bwd_CheckNext )
      wire#w3
      S_Coil( #MB1_Decoder.OpEnabled )
   END_RUNG
   RUNG wire#w2
      Contact( "Decoiler1".Feed.COut.Fwd_CheckNext )
   END_RUNG wire#w3
   RUNG wire#w1
      Contact( "DecoilersHRot".COut.Decoiler1_InLine )
      wire#w4
      Contact( "Decoiler2".Feed.COut.Bwd_CheckNext )
   END_RUNG wire#w3
   RUNG wire#w4
      Contact( "Decoiler2".Feed.COut.Fwd_CheckNext )
   END_RUNG wire#w3
   RUNG wire#w1
      Contact( "DecoilersHRot".COut.Decoiler2_InLine )
      I_Contact( "Decoiler1".Feed.Sts.Standstill )
      wire#w5
      S_Coil( #MB1_Decoder.OpRunning )
   END_RUNG
   RUNG wire#w1
      Contact( "DecoilersHRot".COut.Decoiler1_InLine )
      I_Contact( "Decoiler2".Feed.Sts.Standstill )
   END_RUNG wire#w5
   RUNG wire#w1
      Contact( "Sys".Bit0 )
      S_Coil( #MB1_Decoder.OpDone )
   END_RUNG
   // the same network as SCL:
   #_w1 := #MB1_Decoder.Code = #"1021_DECOILER_OUT_LINE_FEED";
   "A01_HMI".MB1.Button.CoilHandling.Decoiler_OutLine.Feed.Bwd_Minus := #_w1 AND #MB1_Decoder.OperationMinus;
   "A01_HMI".MB1.Button.CoilHandling.Decoiler_OutLine.Feed.Fwd_Plus := #_w1 AND #MB1_Decoder.OperationPlus;
   IF #_w1 AND (("DecoilersHRot".COut.Decoiler2_InLine AND ("Decoiler1".Feed.COut.Bwd_CheckNext OR "Decoiler1".Feed.COut.Fwd_CheckNext)) OR ("DecoilersHRot".COut.Decoiler1_InLine AND ("Decoiler2".Feed.COut.Bwd_CheckNext OR "Decoiler2".Feed.COut.Fwd_CheckNext))) THEN
       #MB1_Decoder.OpEnabled := TRUE;
   END_IF;
   IF #_w1 AND (("DecoilersHRot".COut.Decoiler2_InLine AND NOT "Decoiler1".Feed.Sts.Standstill) OR ("DecoilersHRot".COut.Decoiler1_InLine AND NOT "Decoiler2".Feed.Sts.Standstill)) THEN
       #MB1_Decoder.OpRunning := TRUE;
   END_IF;
   IF #_w1 AND "Sys".Bit0 THEN #MB1_Decoder.OpDone := TRUE; END_IF;
END_REGION

REGION Network 14: MB1 Code 1022 - Decoiler Out Line jaws open / close
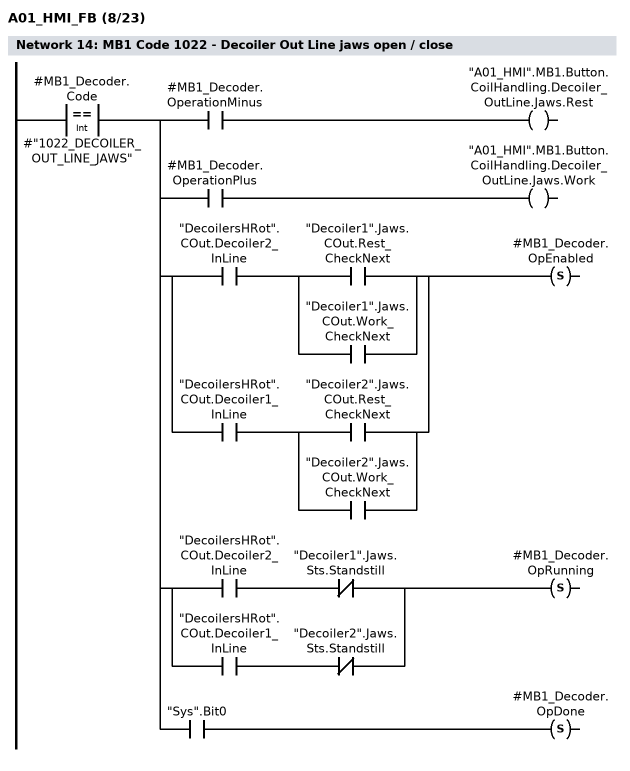
   RUNG wire#powerrail
      { S7_Templates := "SrcType := Int" } EQ_Contact(in1 := #MB1_Decoder.Code, in2 := #"1022_DECOILER_OUT_LINE_JAWS")
      wire#w1
      Contact( #MB1_Decoder.OperationMinus )
      Coil( "A01_HMI".MB1.Button.CoilHandling.Decoiler_OutLine.Jaws.Rest )
   END_RUNG
   RUNG wire#w1
      Contact( #MB1_Decoder.OperationPlus )
      Coil( "A01_HMI".MB1.Button.CoilHandling.Decoiler_OutLine.Jaws.Work )
   END_RUNG
   RUNG wire#w1
      Contact( "DecoilersHRot".COut.Decoiler2_InLine )
      wire#w2
      Contact( "Decoiler1".Jaws.COut.Rest_CheckNext )
      wire#w3
      S_Coil( #MB1_Decoder.OpEnabled )
   END_RUNG
   RUNG wire#w2
      Contact( "Decoiler1".Jaws.COut.Work_CheckNext )
   END_RUNG wire#w3
   RUNG wire#w1
      Contact( "DecoilersHRot".COut.Decoiler1_InLine )
      wire#w4
      Contact( "Decoiler2".Jaws.COut.Rest_CheckNext )
   END_RUNG wire#w3
   RUNG wire#w4
      Contact( "Decoiler2".Jaws.COut.Work_CheckNext )
   END_RUNG wire#w3
   RUNG wire#w1
      Contact( "DecoilersHRot".COut.Decoiler2_InLine )
      I_Contact( "Decoiler1".Jaws.Sts.Standstill )
      wire#w5
      S_Coil( #MB1_Decoder.OpRunning )
   END_RUNG
   RUNG wire#w1
      Contact( "DecoilersHRot".COut.Decoiler1_InLine )
      I_Contact( "Decoiler2".Jaws.Sts.Standstill )
   END_RUNG wire#w5
   RUNG wire#w1
      Contact( "Sys".Bit0 )
      S_Coil( #MB1_Decoder.OpDone )
   END_RUNG
   // the same network as SCL:
   #_w1 := #MB1_Decoder.Code = #"1022_DECOILER_OUT_LINE_JAWS";
   "A01_HMI".MB1.Button.CoilHandling.Decoiler_OutLine.Jaws.Rest := #_w1 AND #MB1_Decoder.OperationMinus;
   "A01_HMI".MB1.Button.CoilHandling.Decoiler_OutLine.Jaws.Work := #_w1 AND #MB1_Decoder.OperationPlus;
   IF #_w1 AND (("DecoilersHRot".COut.Decoiler2_InLine AND ("Decoiler1".Jaws.COut.Rest_CheckNext OR "Decoiler1".Jaws.COut.Work_CheckNext)) OR ("DecoilersHRot".COut.Decoiler1_InLine AND ("Decoiler2".Jaws.COut.Rest_CheckNext OR "Decoiler2".Jaws.COut.Work_CheckNext))) THEN
       #MB1_Decoder.OpEnabled := TRUE;
   END_IF;
   IF #_w1 AND (("DecoilersHRot".COut.Decoiler2_InLine AND NOT "Decoiler1".Jaws.Sts.Standstill) OR ("DecoilersHRot".COut.Decoiler1_InLine AND NOT "Decoiler2".Jaws.Sts.Standstill)) THEN
       #MB1_Decoder.OpRunning := TRUE;
   END_IF;
   IF #_w1 AND "Sys".Bit0 THEN #MB1_Decoder.OpDone := TRUE; END_IF;
END_REGION

REGION Network 15: MB1 Code 1023 - Decoiler Out Line motor coupling rest / work
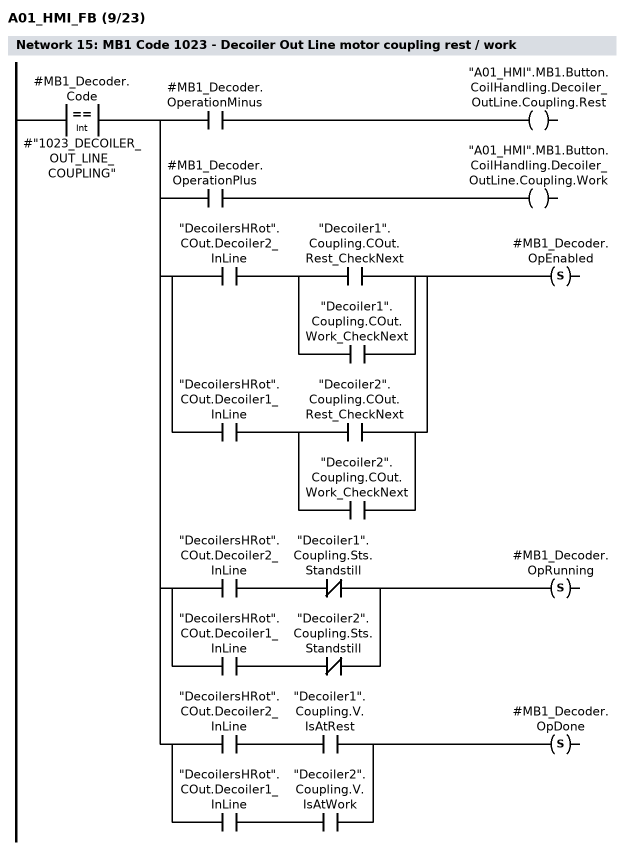
   RUNG wire#powerrail
      { S7_Templates := "SrcType := Int" } EQ_Contact(in1 := #MB1_Decoder.Code, in2 := #"1023_DECOILER_OUT_LINE_COUPLING")
      wire#w1
      Contact( #MB1_Decoder.OperationMinus )
      Coil( "A01_HMI".MB1.Button.CoilHandling.Decoiler_OutLine.Coupling.Rest )
   END_RUNG
   RUNG wire#w1
      Contact( #MB1_Decoder.OperationPlus )
      Coil( "A01_HMI".MB1.Button.CoilHandling.Decoiler_OutLine.Coupling.Work )
   END_RUNG
   RUNG wire#w1
      Contact( "DecoilersHRot".COut.Decoiler2_InLine )
      wire#w2
      Contact( "Decoiler1".Coupling.COut.Rest_CheckNext )
      wire#w3
      S_Coil( #MB1_Decoder.OpEnabled )
   END_RUNG
   RUNG wire#w2
      Contact( "Decoiler1".Coupling.COut.Work_CheckNext )
   END_RUNG wire#w3
   RUNG wire#w1
      Contact( "DecoilersHRot".COut.Decoiler1_InLine )
      wire#w4
      Contact( "Decoiler2".Coupling.COut.Rest_CheckNext )
   END_RUNG wire#w3
   RUNG wire#w4
      Contact( "Decoiler2".Coupling.COut.Work_CheckNext )
   END_RUNG wire#w3
   RUNG wire#w1
      Contact( "DecoilersHRot".COut.Decoiler2_InLine )
      I_Contact( "Decoiler1".Coupling.Sts.Standstill )
      wire#w5
      S_Coil( #MB1_Decoder.OpRunning )
   END_RUNG
   RUNG wire#w1
      Contact( "DecoilersHRot".COut.Decoiler1_InLine )
      I_Contact( "Decoiler2".Coupling.Sts.Standstill )
   END_RUNG wire#w5
   RUNG wire#w1
      Contact( "DecoilersHRot".COut.Decoiler2_InLine )
      Contact( "Decoiler1".Coupling.V.IsAtRest )
      wire#w6
      S_Coil( #MB1_Decoder.OpDone )
   END_RUNG
   RUNG wire#w1
      Contact( "DecoilersHRot".COut.Decoiler1_InLine )
      Contact( "Decoiler2".Coupling.V.IsAtWork )
   END_RUNG wire#w6
   // the same network as SCL:
   #_w1 := #MB1_Decoder.Code = #"1023_DECOILER_OUT_LINE_COUPLING";
   "A01_HMI".MB1.Button.CoilHandling.Decoiler_OutLine.Coupling.Rest := #_w1 AND #MB1_Decoder.OperationMinus;
   "A01_HMI".MB1.Button.CoilHandling.Decoiler_OutLine.Coupling.Work := #_w1 AND #MB1_Decoder.OperationPlus;
   IF #_w1 AND (("DecoilersHRot".COut.Decoiler2_InLine AND ("Decoiler1".Coupling.COut.Rest_CheckNext OR "Decoiler1".Coupling.COut.Work_CheckNext)) OR ("DecoilersHRot".COut.Decoiler1_InLine AND ("Decoiler2".Coupling.COut.Rest_CheckNext OR "Decoiler2".Coupling.COut.Work_CheckNext))) THEN
       #MB1_Decoder.OpEnabled := TRUE;
   END_IF;
   IF #_w1 AND (("DecoilersHRot".COut.Decoiler2_InLine AND NOT "Decoiler1".Coupling.Sts.Standstill) OR ("DecoilersHRot".COut.Decoiler1_InLine AND NOT "Decoiler2".Coupling.Sts.Standstill)) THEN
       #MB1_Decoder.OpRunning := TRUE;
   END_IF;
   IF #_w1 AND (("DecoilersHRot".COut.Decoiler2_InLine AND "Decoiler1".Coupling.V.IsAtRest) OR ("DecoilersHRot".COut.Decoiler1_InLine AND "Decoiler2".Coupling.V.IsAtWork)) THEN
       #MB1_Decoder.OpDone := TRUE;
   END_IF;
END_REGION

REGION Network 16: MB1 Code 1024 - Decoiler Out Line snubber lift up / down
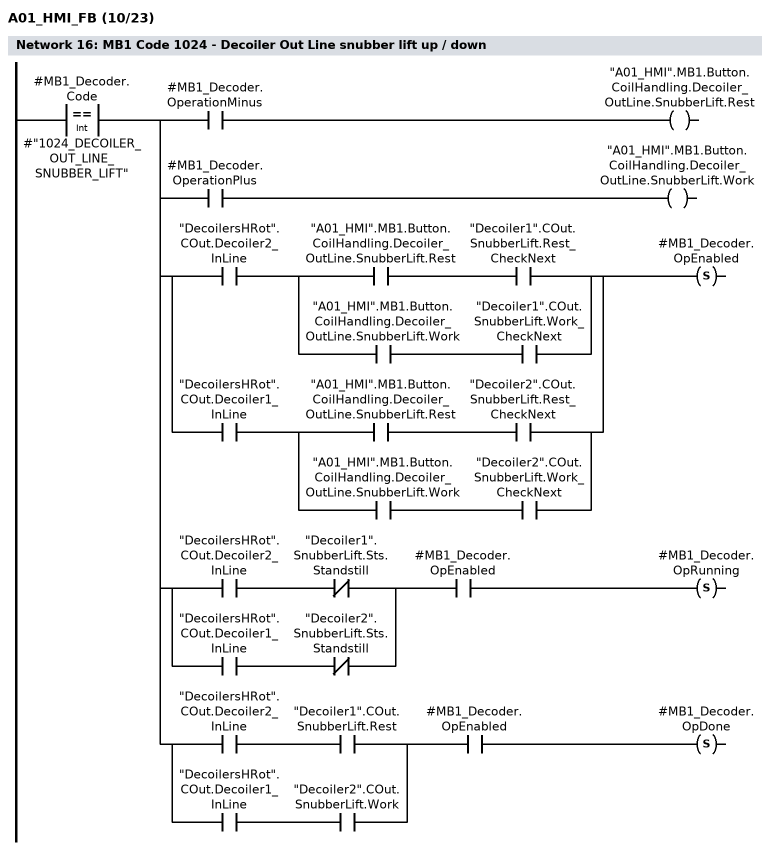
   RUNG wire#powerrail
      { S7_Templates := "SrcType := Int" } EQ_Contact(in1 := #MB1_Decoder.Code, in2 := #"1024_DECOILER_OUT_LINE_SNUBBER_LIFT")
      wire#w1
      Contact( #MB1_Decoder.OperationMinus )
      Coil( "A01_HMI".MB1.Button.CoilHandling.Decoiler_OutLine.SnubberLift.Rest )
   END_RUNG
   RUNG wire#w1
      Contact( #MB1_Decoder.OperationPlus )
      Coil( "A01_HMI".MB1.Button.CoilHandling.Decoiler_OutLine.SnubberLift.Work )
   END_RUNG
   RUNG wire#w1
      Contact( "DecoilersHRot".COut.Decoiler2_InLine )
      wire#w2
      Contact( "A01_HMI".MB1.Button.CoilHandling.Decoiler_OutLine.SnubberLift.Rest )
      Contact( "Decoiler1".COut.SnubberLift.Rest_CheckNext )
      wire#w3
      S_Coil( #MB1_Decoder.OpEnabled )
   END_RUNG
   RUNG wire#w2
      Contact( "A01_HMI".MB1.Button.CoilHandling.Decoiler_OutLine.SnubberLift.Work )
      Contact( "Decoiler1".COut.SnubberLift.Work_CheckNext )
   END_RUNG wire#w3
   RUNG wire#w1
      Contact( "DecoilersHRot".COut.Decoiler1_InLine )
      wire#w4
      Contact( "A01_HMI".MB1.Button.CoilHandling.Decoiler_OutLine.SnubberLift.Rest )
      Contact( "Decoiler2".COut.SnubberLift.Rest_CheckNext )
   END_RUNG wire#w3
   RUNG wire#w4
      Contact( "A01_HMI".MB1.Button.CoilHandling.Decoiler_OutLine.SnubberLift.Work )
      Contact( "Decoiler2".COut.SnubberLift.Work_CheckNext )
   END_RUNG wire#w3
   RUNG wire#w1
      Contact( "DecoilersHRot".COut.Decoiler2_InLine )
      I_Contact( "Decoiler1".SnubberLift.Sts.Standstill )
      wire#w5
      Contact( #MB1_Decoder.OpEnabled )
      S_Coil( #MB1_Decoder.OpRunning )
   END_RUNG
   RUNG wire#w1
      Contact( "DecoilersHRot".COut.Decoiler1_InLine )
      I_Contact( "Decoiler2".SnubberLift.Sts.Standstill )
   END_RUNG wire#w5
   RUNG wire#w1
      Contact( "DecoilersHRot".COut.Decoiler2_InLine )
      Contact( "Decoiler1".COut.SnubberLift.Rest )
      wire#w6
      Contact( #MB1_Decoder.OpEnabled )
      S_Coil( #MB1_Decoder.OpDone )
   END_RUNG
   RUNG wire#w1
      Contact( "DecoilersHRot".COut.Decoiler1_InLine )
      Contact( "Decoiler2".COut.SnubberLift.Work )
   END_RUNG wire#w6
   // the same network as SCL:
   #_w1 := #MB1_Decoder.Code = #"1024_DECOILER_OUT_LINE_SNUBBER_LIFT";
   "A01_HMI".MB1.Button.CoilHandling.Decoiler_OutLine.SnubberLift.Rest := #_w1 AND #MB1_Decoder.OperationMinus;
   "A01_HMI".MB1.Button.CoilHandling.Decoiler_OutLine.SnubberLift.Work := #_w1 AND #MB1_Decoder.OperationPlus;
   IF #_w1 AND (("DecoilersHRot".COut.Decoiler2_InLine AND (("A01_HMI".MB1.Button.CoilHandling.Decoiler_OutLine.SnubberLift.Rest AND "Decoiler1".COut.SnubberLift.Rest_CheckNext) OR ("A01_HMI".MB1.Button.CoilHandling.Decoiler_OutLine.SnubberLift.Work AND "Decoiler1".COut.SnubberLift.Work_CheckNext))) OR ("DecoilersHRot".COut.Decoiler1_InLine AND (("A01_HMI".MB1.Button.CoilHandling.Decoiler_OutLine.SnubberLift.Rest AND "Decoiler2".COut.SnubberLift.Rest_CheckNext) OR ("A01_HMI".MB1.Button.CoilHandling.Decoiler_OutLine.SnubberLift.Work AND "Decoiler2".COut.SnubberLift.Work_CheckNext)))) THEN
       #MB1_Decoder.OpEnabled := TRUE;
   END_IF;
   IF #_w1 AND (("DecoilersHRot".COut.Decoiler2_InLine AND NOT "Decoiler1".SnubberLift.Sts.Standstill) OR ("DecoilersHRot".COut.Decoiler1_InLine AND NOT "Decoiler2".SnubberLift.Sts.Standstill)) AND #MB1_Decoder.OpEnabled THEN
       #MB1_Decoder.OpRunning := TRUE;
   END_IF;
   IF #_w1 AND (("DecoilersHRot".COut.Decoiler2_InLine AND "Decoiler1".COut.SnubberLift.Rest) OR ("DecoilersHRot".COut.Decoiler1_InLine AND "Decoiler2".COut.SnubberLift.Work)) AND #MB1_Decoder.OpEnabled THEN
       #MB1_Decoder.OpDone := TRUE;
   END_IF;
END_REGION

REGION Network 17: MB1 Code 1025 - Decoiler Out Line nubber roll bkw / fwd
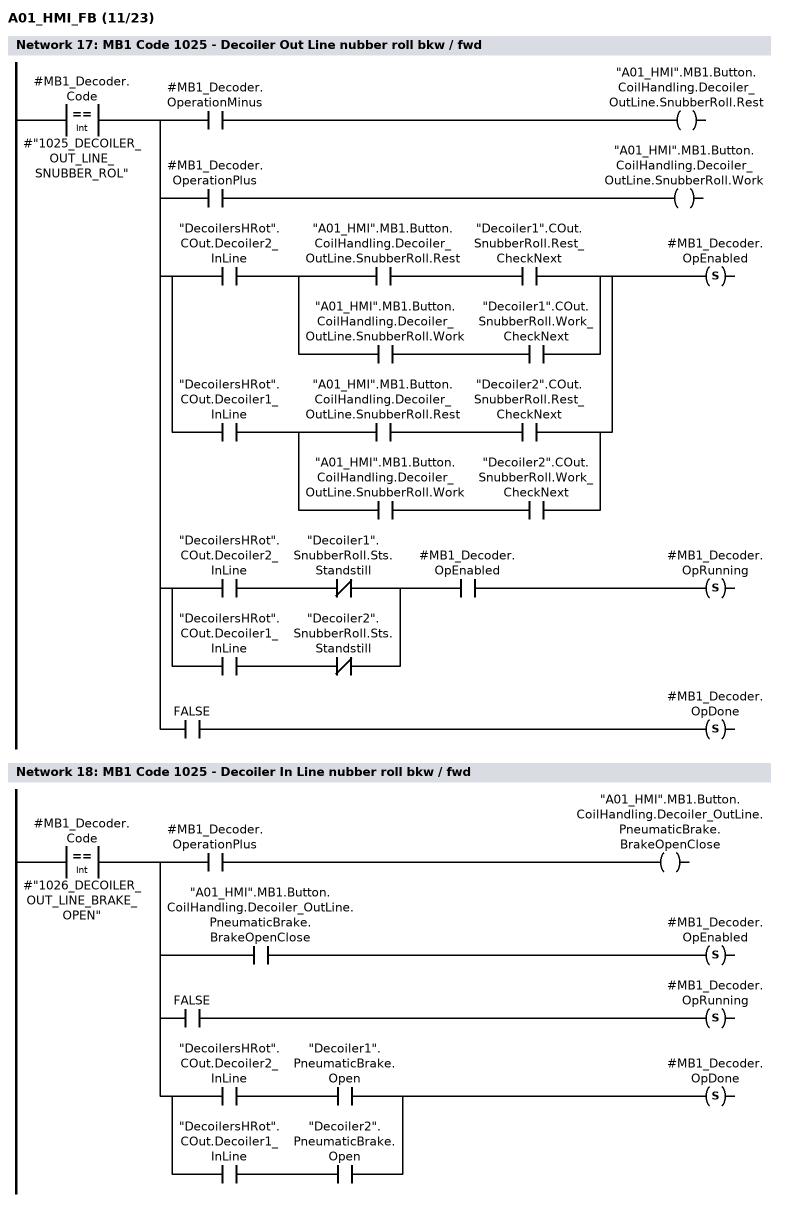
   RUNG wire#powerrail
      { S7_Templates := "SrcType := Int" } EQ_Contact(in1 := #MB1_Decoder.Code, in2 := #"1025_DECOILER_OUT_LINE_SNUBBER_ROL")
      wire#w1
      Contact( #MB1_Decoder.OperationMinus )
      Coil( "A01_HMI".MB1.Button.CoilHandling.Decoiler_OutLine.SnubberRoll.Rest )
   END_RUNG
   RUNG wire#w1
      Contact( #MB1_Decoder.OperationPlus )
      Coil( "A01_HMI".MB1.Button.CoilHandling.Decoiler_OutLine.SnubberRoll.Work )
   END_RUNG
   RUNG wire#w1
      Contact( "DecoilersHRot".COut.Decoiler2_InLine )
      wire#w2
      Contact( "A01_HMI".MB1.Button.CoilHandling.Decoiler_OutLine.SnubberRoll.Rest )
      Contact( "Decoiler1".COut.SnubberRoll.Rest_CheckNext )
      wire#w3
      S_Coil( #MB1_Decoder.OpEnabled )
   END_RUNG
   RUNG wire#w2
      Contact( "A01_HMI".MB1.Button.CoilHandling.Decoiler_OutLine.SnubberRoll.Work )
      Contact( "Decoiler1".COut.SnubberRoll.Work_CheckNext )
   END_RUNG wire#w3
   RUNG wire#w1
      Contact( "DecoilersHRot".COut.Decoiler1_InLine )
      wire#w4
      Contact( "A01_HMI".MB1.Button.CoilHandling.Decoiler_OutLine.SnubberRoll.Rest )
      Contact( "Decoiler2".COut.SnubberRoll.Rest_CheckNext )
   END_RUNG wire#w3
   RUNG wire#w4
      Contact( "A01_HMI".MB1.Button.CoilHandling.Decoiler_OutLine.SnubberRoll.Work )
      Contact( "Decoiler2".COut.SnubberRoll.Work_CheckNext )
   END_RUNG wire#w3
   RUNG wire#w1
      Contact( "DecoilersHRot".COut.Decoiler2_InLine )
      I_Contact( "Decoiler1".SnubberRoll.Sts.Standstill )
      wire#w5
      Contact( #MB1_Decoder.OpEnabled )
      S_Coil( #MB1_Decoder.OpRunning )
   END_RUNG
   RUNG wire#w1
      Contact( "DecoilersHRot".COut.Decoiler1_InLine )
      I_Contact( "Decoiler2".SnubberRoll.Sts.Standstill )
   END_RUNG wire#w5
   RUNG wire#w1
      Contact( FALSE )
      S_Coil( #MB1_Decoder.OpDone )
   END_RUNG
   // the same network as SCL:
   #_w1 := #MB1_Decoder.Code = #"1025_DECOILER_OUT_LINE_SNUBBER_ROL";
   "A01_HMI".MB1.Button.CoilHandling.Decoiler_OutLine.SnubberRoll.Rest := #_w1 AND #MB1_Decoder.OperationMinus;
   "A01_HMI".MB1.Button.CoilHandling.Decoiler_OutLine.SnubberRoll.Work := #_w1 AND #MB1_Decoder.OperationPlus;
   IF #_w1 AND (("DecoilersHRot".COut.Decoiler2_InLine AND (("A01_HMI".MB1.Button.CoilHandling.Decoiler_OutLine.SnubberRoll.Rest AND "Decoiler1".COut.SnubberRoll.Rest_CheckNext) OR ("A01_HMI".MB1.Button.CoilHandling.Decoiler_OutLine.SnubberRoll.Work AND "Decoiler1".COut.SnubberRoll.Work_CheckNext))) OR ("DecoilersHRot".COut.Decoiler1_InLine AND (("A01_HMI".MB1.Button.CoilHandling.Decoiler_OutLine.SnubberRoll.Rest AND "Decoiler2".COut.SnubberRoll.Rest_CheckNext) OR ("A01_HMI".MB1.Button.CoilHandling.Decoiler_OutLine.SnubberRoll.Work AND "Decoiler2".COut.SnubberRoll.Work_CheckNext)))) THEN
       #MB1_Decoder.OpEnabled := TRUE;
   END_IF;
   IF #_w1 AND (("DecoilersHRot".COut.Decoiler2_InLine AND NOT "Decoiler1".SnubberRoll.Sts.Standstill) OR ("DecoilersHRot".COut.Decoiler1_InLine AND NOT "Decoiler2".SnubberRoll.Sts.Standstill)) AND #MB1_Decoder.OpEnabled THEN
       #MB1_Decoder.OpRunning := TRUE;
   END_IF;
   IF #_w1 AND FALSE THEN #MB1_Decoder.OpDone := TRUE; END_IF;
END_REGION

REGION Network 18: MB1 Code 1025 - Decoiler In Line nubber roll bkw / fwd
   RUNG wire#powerrail
      { S7_Templates := "SrcType := Int" } EQ_Contact(in1 := #MB1_Decoder.Code, in2 := #"1026_DECOILER_OUT_LINE_BRAKE_OPEN")
      wire#w1
      Contact( #MB1_Decoder.OperationPlus )
      Coil( "A01_HMI".MB1.Button.CoilHandling.Decoiler_OutLine.PneumaticBrake.BrakeOpenClose )
   END_RUNG
   RUNG wire#w1
      Contact( "A01_HMI".MB1.Button.CoilHandling.Decoiler_OutLine.PneumaticBrake.BrakeOpenClose )
      S_Coil( #MB1_Decoder.OpEnabled )
   END_RUNG
   RUNG wire#w1
      Contact( FALSE )
      S_Coil( #MB1_Decoder.OpRunning )
   END_RUNG
   RUNG wire#w1
      Contact( "DecoilersHRot".COut.Decoiler2_InLine )
      Contact( "Decoiler1".PneumaticBrake.Open )
      wire#w2
      S_Coil( #MB1_Decoder.OpDone )
   END_RUNG
   RUNG wire#w1
      Contact( "DecoilersHRot".COut.Decoiler1_InLine )
      Contact( "Decoiler2".PneumaticBrake.Open )
   END_RUNG wire#w2
   // the same network as SCL:
   #_w1 := #MB1_Decoder.Code = #"1026_DECOILER_OUT_LINE_BRAKE_OPEN";
   "A01_HMI".MB1.Button.CoilHandling.Decoiler_OutLine.PneumaticBrake.BrakeOpenClose := #_w1 AND #MB1_Decoder.OperationPlus;
   IF #_w1 AND "A01_HMI".MB1.Button.CoilHandling.Decoiler_OutLine.PneumaticBrake.BrakeOpenClose THEN
       #MB1_Decoder.OpEnabled := TRUE;
   END_IF;
   IF #_w1 AND FALSE THEN #MB1_Decoder.OpRunning := TRUE; END_IF;
   IF #_w1 AND (("DecoilersHRot".COut.Decoiler2_InLine AND "Decoiler1".PneumaticBrake.Open) OR ("DecoilersHRot".COut.Decoiler1_InLine AND "Decoiler2".PneumaticBrake.Open)) THEN
       #MB1_Decoder.OpDone := TRUE;
   END_IF;
END_REGION

REGION Network 19: MB1 Code 1017 - Decoiler In Line pneumatic brake partial
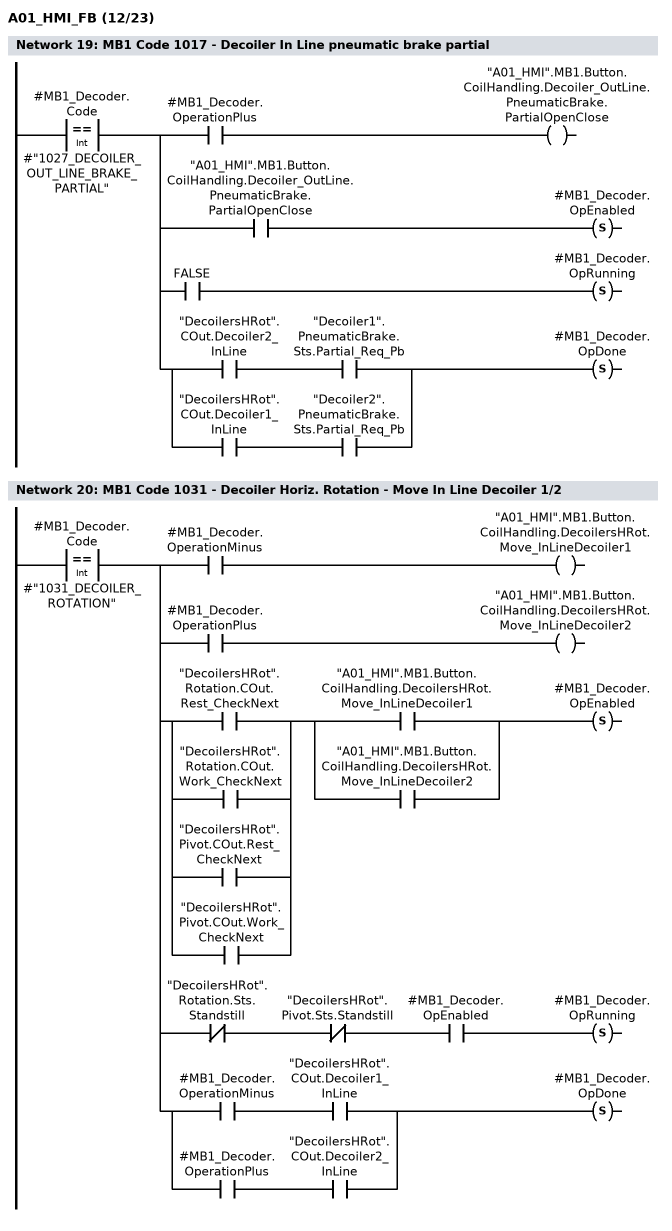
   RUNG wire#powerrail
      { S7_Templates := "SrcType := Int" } EQ_Contact(in1 := #MB1_Decoder.Code, in2 := #"1027_DECOILER_OUT_LINE_BRAKE_PARTIAL")
      wire#w1
      Contact( #MB1_Decoder.OperationPlus )
      Coil( "A01_HMI".MB1.Button.CoilHandling.Decoiler_OutLine.PneumaticBrake.PartialOpenClose )
   END_RUNG
   RUNG wire#w1
      Contact( "A01_HMI".MB1.Button.CoilHandling.Decoiler_OutLine.PneumaticBrake.PartialOpenClose )
      S_Coil( #MB1_Decoder.OpEnabled )
   END_RUNG
   RUNG wire#w1
      Contact( FALSE )
      S_Coil( #MB1_Decoder.OpRunning )
   END_RUNG
   RUNG wire#w1
      Contact( "DecoilersHRot".COut.Decoiler2_InLine )
      Contact( "Decoiler1".PneumaticBrake.Sts.Partial_Req_Pb )
      wire#w2
      S_Coil( #MB1_Decoder.OpDone )
   END_RUNG
   RUNG wire#w1
      Contact( "DecoilersHRot".COut.Decoiler1_InLine )
      Contact( "Decoiler2".PneumaticBrake.Sts.Partial_Req_Pb )
   END_RUNG wire#w2
   // the same network as SCL:
   #_w1 := #MB1_Decoder.Code = #"1027_DECOILER_OUT_LINE_BRAKE_PARTIAL";
   "A01_HMI".MB1.Button.CoilHandling.Decoiler_OutLine.PneumaticBrake.PartialOpenClose := #_w1 AND #MB1_Decoder.OperationPlus;
   IF #_w1 AND "A01_HMI".MB1.Button.CoilHandling.Decoiler_OutLine.PneumaticBrake.PartialOpenClose THEN
       #MB1_Decoder.OpEnabled := TRUE;
   END_IF;
   IF #_w1 AND FALSE THEN #MB1_Decoder.OpRunning := TRUE; END_IF;
   IF #_w1 AND (("DecoilersHRot".COut.Decoiler2_InLine AND "Decoiler1".PneumaticBrake.Sts.Partial_Req_Pb) OR ("DecoilersHRot".COut.Decoiler1_InLine AND "Decoiler2".PneumaticBrake.Sts.Partial_Req_Pb)) THEN
       #MB1_Decoder.OpDone := TRUE;
   END_IF;
END_REGION

REGION Network 20: MB1 Code 1031 - Decoiler Horiz. Rotation - Move In Line Decoiler 1/2
   RUNG wire#powerrail
      { S7_Templates := "SrcType := Int" } EQ_Contact(in1 := #MB1_Decoder.Code, in2 := #"1031_DECOILER_ROTATION")
      wire#w1
      Contact( #MB1_Decoder.OperationMinus )
      Coil( "A01_HMI".MB1.Button.CoilHandling.DecoilersHRot.Move_InLineDecoiler1 )
   END_RUNG
   RUNG wire#w1
      Contact( #MB1_Decoder.OperationPlus )
      Coil( "A01_HMI".MB1.Button.CoilHandling.DecoilersHRot.Move_InLineDecoiler2 )
   END_RUNG
   RUNG wire#w1
      Contact( "DecoilersHRot".Rotation.COut.Rest_CheckNext )
      wire#w2
      Contact( "A01_HMI".MB1.Button.CoilHandling.DecoilersHRot.Move_InLineDecoiler1 )
      wire#w3
      S_Coil( #MB1_Decoder.OpEnabled )
   END_RUNG
   RUNG wire#w1
      Contact( "DecoilersHRot".Rotation.COut.Work_CheckNext )
   END_RUNG wire#w2
   RUNG wire#w1
      Contact( "DecoilersHRot".Pivot.COut.Rest_CheckNext )
   END_RUNG wire#w2
   RUNG wire#w1
      Contact( "DecoilersHRot".Pivot.COut.Work_CheckNext )
   END_RUNG wire#w2
   RUNG wire#w2
      Contact( "A01_HMI".MB1.Button.CoilHandling.DecoilersHRot.Move_InLineDecoiler2 )
   END_RUNG wire#w3
   RUNG wire#w1
      I_Contact( "DecoilersHRot".Rotation.Sts.Standstill )
      I_Contact( "DecoilersHRot".Pivot.Sts.Standstill )
      Contact( #MB1_Decoder.OpEnabled )
      S_Coil( #MB1_Decoder.OpRunning )
   END_RUNG
   RUNG wire#w1
      Contact( #MB1_Decoder.OperationMinus )
      Contact( "DecoilersHRot".COut.Decoiler1_InLine )
      wire#w4
      S_Coil( #MB1_Decoder.OpDone )
   END_RUNG
   RUNG wire#w1
      Contact( #MB1_Decoder.OperationPlus )
      Contact( "DecoilersHRot".COut.Decoiler2_InLine )
   END_RUNG wire#w4
   // the same network as SCL:
   #_w1 := #MB1_Decoder.Code = #"1031_DECOILER_ROTATION";
   "A01_HMI".MB1.Button.CoilHandling.DecoilersHRot.Move_InLineDecoiler1 := #_w1 AND #MB1_Decoder.OperationMinus;
   "A01_HMI".MB1.Button.CoilHandling.DecoilersHRot.Move_InLineDecoiler2 := #_w1 AND #MB1_Decoder.OperationPlus;
   IF #_w1 AND ("DecoilersHRot".Rotation.COut.Rest_CheckNext OR "DecoilersHRot".Rotation.COut.Work_CheckNext OR "DecoilersHRot".Pivot.COut.Rest_CheckNext OR "DecoilersHRot".Pivot.COut.Work_CheckNext) AND ("A01_HMI".MB1.Button.CoilHandling.DecoilersHRot.Move_InLineDecoiler1 OR "A01_HMI".MB1.Button.CoilHandling.DecoilersHRot.Move_InLineDecoiler2) THEN
       #MB1_Decoder.OpEnabled := TRUE;
   END_IF;
   IF #_w1 AND NOT "DecoilersHRot".Rotation.Sts.Standstill AND NOT "DecoilersHRot".Pivot.Sts.Standstill AND #MB1_Decoder.OpEnabled THEN
       #MB1_Decoder.OpRunning := TRUE;
   END_IF;
   IF #_w1 AND ((#MB1_Decoder.OperationMinus AND "DecoilersHRot".COut.Decoiler1_InLine) OR (#MB1_Decoder.OperationPlus AND "DecoilersHRot".COut.Decoiler2_InLine)) THEN
       #MB1_Decoder.OpDone := TRUE;
   END_IF;
END_REGION

REGION Network 21: MB1 Code 1032 - Decoiler Rotation In Line Direction
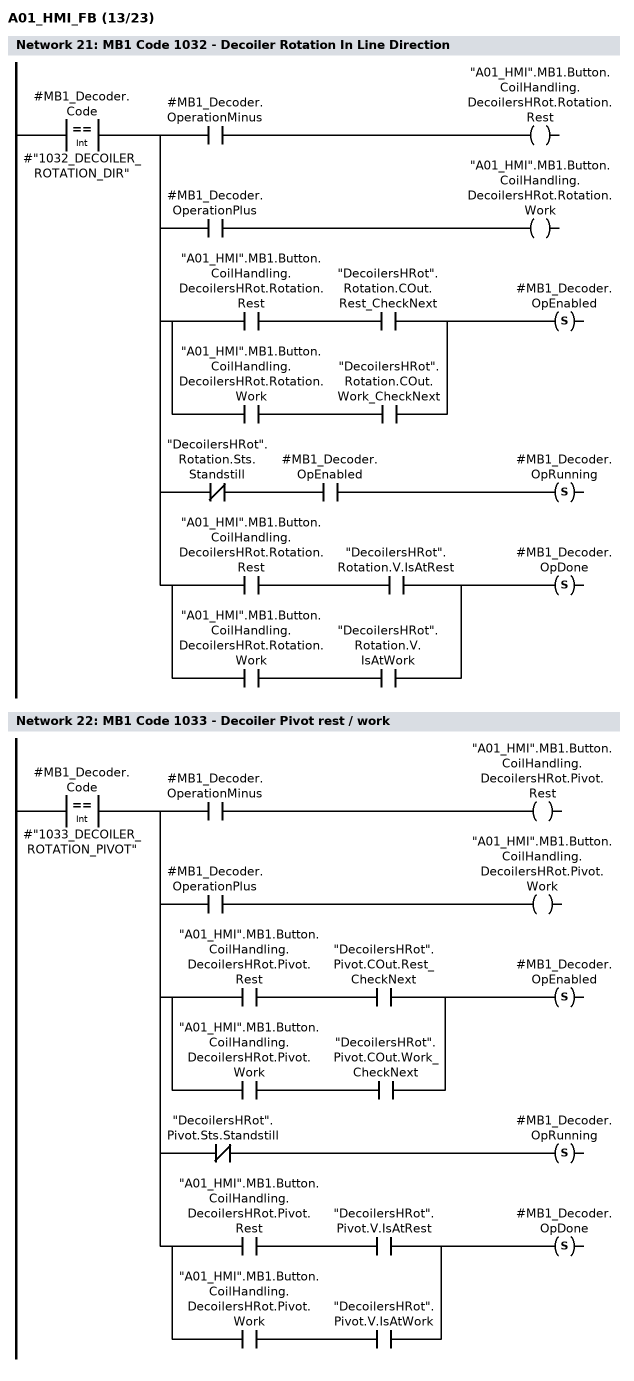
   RUNG wire#powerrail
      { S7_Templates := "SrcType := Int" } EQ_Contact(in1 := #MB1_Decoder.Code, in2 := #"1032_DECOILER_ROTATION_DIR")
      wire#w1
      Contact( #MB1_Decoder.OperationMinus )
      Coil( "A01_HMI".MB1.Button.CoilHandling.DecoilersHRot.Rotation.Rest )
   END_RUNG
   RUNG wire#w1
      Contact( #MB1_Decoder.OperationPlus )
      Coil( "A01_HMI".MB1.Button.CoilHandling.DecoilersHRot.Rotation.Work )
   END_RUNG
   RUNG wire#w1
      Contact( "A01_HMI".MB1.Button.CoilHandling.DecoilersHRot.Rotation.Rest )
      Contact( "DecoilersHRot".Rotation.COut.Rest_CheckNext )
      wire#w2
      S_Coil( #MB1_Decoder.OpEnabled )
   END_RUNG
   RUNG wire#w1
      Contact( "A01_HMI".MB1.Button.CoilHandling.DecoilersHRot.Rotation.Work )
      Contact( "DecoilersHRot".Rotation.COut.Work_CheckNext )
   END_RUNG wire#w2
   RUNG wire#w1
      I_Contact( "DecoilersHRot".Rotation.Sts.Standstill )
      Contact( #MB1_Decoder.OpEnabled )
      S_Coil( #MB1_Decoder.OpRunning )
   END_RUNG
   RUNG wire#w1
      Contact( "A01_HMI".MB1.Button.CoilHandling.DecoilersHRot.Rotation.Rest )
      Contact( "DecoilersHRot".Rotation.V.IsAtRest )
      wire#w3
      S_Coil( #MB1_Decoder.OpDone )
   END_RUNG
   RUNG wire#w1
      Contact( "A01_HMI".MB1.Button.CoilHandling.DecoilersHRot.Rotation.Work )
      Contact( "DecoilersHRot".Rotation.V.IsAtWork )
   END_RUNG wire#w3
   // the same network as SCL:
   #_w1 := #MB1_Decoder.Code = #"1032_DECOILER_ROTATION_DIR";
   "A01_HMI".MB1.Button.CoilHandling.DecoilersHRot.Rotation.Rest := #_w1 AND #MB1_Decoder.OperationMinus;
   "A01_HMI".MB1.Button.CoilHandling.DecoilersHRot.Rotation.Work := #_w1 AND #MB1_Decoder.OperationPlus;
   IF #_w1 AND (("A01_HMI".MB1.Button.CoilHandling.DecoilersHRot.Rotation.Rest AND "DecoilersHRot".Rotation.COut.Rest_CheckNext) OR ("A01_HMI".MB1.Button.CoilHandling.DecoilersHRot.Rotation.Work AND "DecoilersHRot".Rotation.COut.Work_CheckNext)) THEN
       #MB1_Decoder.OpEnabled := TRUE;
   END_IF;
   IF #_w1 AND NOT "DecoilersHRot".Rotation.Sts.Standstill AND #MB1_Decoder.OpEnabled THEN
       #MB1_Decoder.OpRunning := TRUE;
   END_IF;
   IF #_w1 AND (("A01_HMI".MB1.Button.CoilHandling.DecoilersHRot.Rotation.Rest AND "DecoilersHRot".Rotation.V.IsAtRest) OR ("A01_HMI".MB1.Button.CoilHandling.DecoilersHRot.Rotation.Work AND "DecoilersHRot".Rotation.V.IsAtWork)) THEN
       #MB1_Decoder.OpDone := TRUE;
   END_IF;
END_REGION

REGION Network 22: MB1 Code 1033 - Decoiler Pivot rest / work
   RUNG wire#powerrail
      { S7_Templates := "SrcType := Int" } EQ_Contact(in1 := #MB1_Decoder.Code, in2 := #"1033_DECOILER_ROTATION_PIVOT")
      wire#w1
      Contact( #MB1_Decoder.OperationMinus )
      Coil( "A01_HMI".MB1.Button.CoilHandling.DecoilersHRot.Pivot.Rest )
   END_RUNG
   RUNG wire#w1
      Contact( #MB1_Decoder.OperationPlus )
      Coil( "A01_HMI".MB1.Button.CoilHandling.DecoilersHRot.Pivot.Work )
   END_RUNG
   RUNG wire#w1
      Contact( "A01_HMI".MB1.Button.CoilHandling.DecoilersHRot.Pivot.Rest )
      Contact( "DecoilersHRot".Pivot.COut.Rest_CheckNext )
      wire#w2
      S_Coil( #MB1_Decoder.OpEnabled )
   END_RUNG
   RUNG wire#w1
      Contact( "A01_HMI".MB1.Button.CoilHandling.DecoilersHRot.Pivot.Work )
      Contact( "DecoilersHRot".Pivot.COut.Work_CheckNext )
   END_RUNG wire#w2
   RUNG wire#w1
      I_Contact( "DecoilersHRot".Pivot.Sts.Standstill )
      S_Coil( #MB1_Decoder.OpRunning )
   END_RUNG
   RUNG wire#w1
      Contact( "A01_HMI".MB1.Button.CoilHandling.DecoilersHRot.Pivot.Rest )
      Contact( "DecoilersHRot".Pivot.V.IsAtRest )
      wire#w3
      S_Coil( #MB1_Decoder.OpDone )
   END_RUNG
   RUNG wire#w1
      Contact( "A01_HMI".MB1.Button.CoilHandling.DecoilersHRot.Pivot.Work )
      Contact( "DecoilersHRot".Pivot.V.IsAtWork )
   END_RUNG wire#w3
   // the same network as SCL:
   #_w1 := #MB1_Decoder.Code = #"1033_DECOILER_ROTATION_PIVOT";
   "A01_HMI".MB1.Button.CoilHandling.DecoilersHRot.Pivot.Rest := #_w1 AND #MB1_Decoder.OperationMinus;
   "A01_HMI".MB1.Button.CoilHandling.DecoilersHRot.Pivot.Work := #_w1 AND #MB1_Decoder.OperationPlus;
   IF #_w1 AND (("A01_HMI".MB1.Button.CoilHandling.DecoilersHRot.Pivot.Rest AND "DecoilersHRot".Pivot.COut.Rest_CheckNext) OR ("A01_HMI".MB1.Button.CoilHandling.DecoilersHRot.Pivot.Work AND "DecoilersHRot".Pivot.COut.Work_CheckNext)) THEN
       #MB1_Decoder.OpEnabled := TRUE;
   END_IF;
   IF #_w1 AND NOT "DecoilersHRot".Pivot.Sts.Standstill THEN #MB1_Decoder.OpRunning := TRUE; END_IF;
   IF #_w1 AND (("A01_HMI".MB1.Button.CoilHandling.DecoilersHRot.Pivot.Rest AND "DecoilersHRot".Pivot.V.IsAtRest) OR ("A01_HMI".MB1.Button.CoilHandling.DecoilersHRot.Pivot.Work AND "DecoilersHRot".Pivot.V.IsAtWork)) THEN
       #MB1_Decoder.OpDone := TRUE;
   END_IF;
END_REGION

REGION Network 23: MB1 Code 1034 - Decoiler traslation BWD / FWD
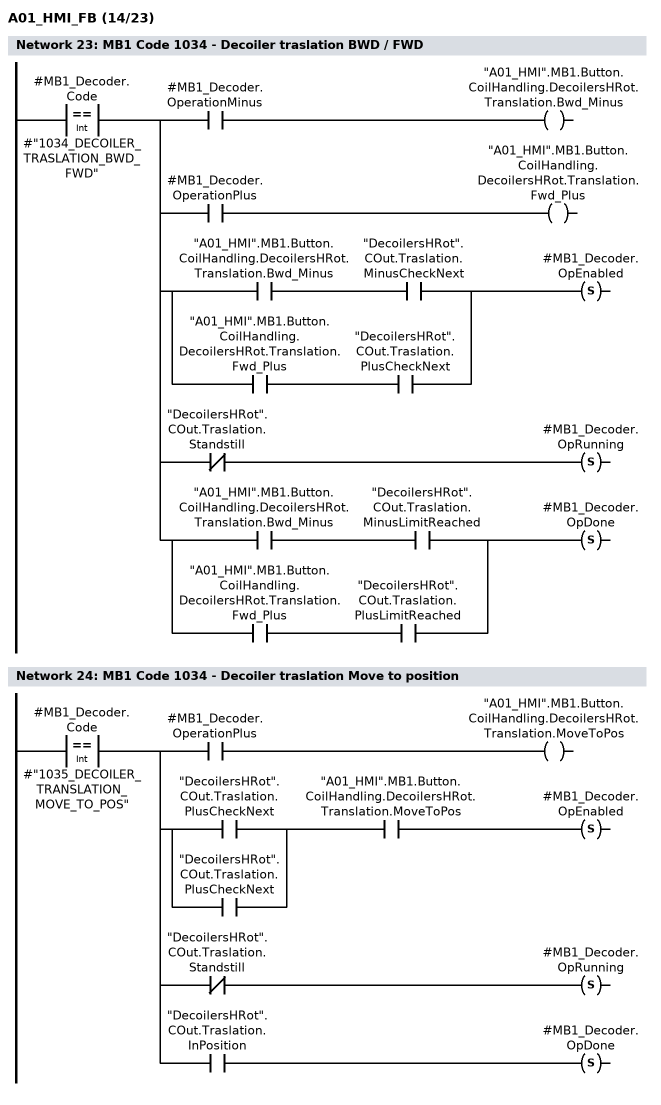
   RUNG wire#powerrail
      { S7_Templates := "SrcType := Int" } EQ_Contact(in1 := #MB1_Decoder.Code, in2 := #"1034_DECOILER_TRASLATION_BWD_FWD")
      wire#w1
      Contact( #MB1_Decoder.OperationMinus )
      Coil( "A01_HMI".MB1.Button.CoilHandling.DecoilersHRot.Translation.Bwd_Minus )
   END_RUNG
   RUNG wire#w1
      Contact( #MB1_Decoder.OperationPlus )
      Coil( "A01_HMI".MB1.Button.CoilHandling.DecoilersHRot.Translation.Fwd_Plus )
   END_RUNG
   RUNG wire#w1
      Contact( "A01_HMI".MB1.Button.CoilHandling.DecoilersHRot.Translation.Bwd_Minus )
      Contact( "DecoilersHRot".COut.Traslation.MinusCheckNext )
      wire#w2
      S_Coil( #MB1_Decoder.OpEnabled )
   END_RUNG
   RUNG wire#w1
      Contact( "A01_HMI".MB1.Button.CoilHandling.DecoilersHRot.Translation.Fwd_Plus )
      Contact( "DecoilersHRot".COut.Traslation.PlusCheckNext )
   END_RUNG wire#w2
   RUNG wire#w1
      I_Contact( "DecoilersHRot".COut.Traslation.Standstill )
      S_Coil( #MB1_Decoder.OpRunning )
   END_RUNG
   RUNG wire#w1
      Contact( "A01_HMI".MB1.Button.CoilHandling.DecoilersHRot.Translation.Bwd_Minus )
      Contact( "DecoilersHRot".COut.Traslation.MinusLimitReached )
      wire#w3
      S_Coil( #MB1_Decoder.OpDone )
   END_RUNG
   RUNG wire#w1
      Contact( "A01_HMI".MB1.Button.CoilHandling.DecoilersHRot.Translation.Fwd_Plus )
      Contact( "DecoilersHRot".COut.Traslation.PlusLimitReached )
   END_RUNG wire#w3
   // the same network as SCL:
   #_w1 := #MB1_Decoder.Code = #"1034_DECOILER_TRASLATION_BWD_FWD";
   "A01_HMI".MB1.Button.CoilHandling.DecoilersHRot.Translation.Bwd_Minus := #_w1 AND #MB1_Decoder.OperationMinus;
   "A01_HMI".MB1.Button.CoilHandling.DecoilersHRot.Translation.Fwd_Plus := #_w1 AND #MB1_Decoder.OperationPlus;
   IF #_w1 AND (("A01_HMI".MB1.Button.CoilHandling.DecoilersHRot.Translation.Bwd_Minus AND "DecoilersHRot".COut.Traslation.MinusCheckNext) OR ("A01_HMI".MB1.Button.CoilHandling.DecoilersHRot.Translation.Fwd_Plus AND "DecoilersHRot".COut.Traslation.PlusCheckNext)) THEN
       #MB1_Decoder.OpEnabled := TRUE;
   END_IF;
   IF #_w1 AND NOT "DecoilersHRot".COut.Traslation.Standstill THEN #MB1_Decoder.OpRunning := TRUE; END_IF;
   IF #_w1 AND (("A01_HMI".MB1.Button.CoilHandling.DecoilersHRot.Translation.Bwd_Minus AND "DecoilersHRot".COut.Traslation.MinusLimitReached) OR ("A01_HMI".MB1.Button.CoilHandling.DecoilersHRot.Translation.Fwd_Plus AND "DecoilersHRot".COut.Traslation.PlusLimitReached)) THEN
       #MB1_Decoder.OpDone := TRUE;
   END_IF;
END_REGION

REGION Network 24: MB1 Code 1034 - Decoiler traslation Move to position
   RUNG wire#powerrail
      { S7_Templates := "SrcType := Int" } EQ_Contact(in1 := #MB1_Decoder.Code, in2 := #"1035_DECOILER_TRANSLATION_MOVE_TO_POS")
      wire#w1
      Contact( #MB1_Decoder.OperationPlus )
      Coil( "A01_HMI".MB1.Button.CoilHandling.DecoilersHRot.Translation.MoveToPos )
   END_RUNG
   RUNG wire#w1
      Contact( "DecoilersHRot".COut.Traslation.PlusCheckNext )
      wire#w2
      Contact( "A01_HMI".MB1.Button.CoilHandling.DecoilersHRot.Translation.MoveToPos )
      S_Coil( #MB1_Decoder.OpEnabled )
   END_RUNG
   RUNG wire#w1
      Contact( "DecoilersHRot".COut.Traslation.PlusCheckNext )
   END_RUNG wire#w2
   RUNG wire#w1
      I_Contact( "DecoilersHRot".COut.Traslation.Standstill )
      S_Coil( #MB1_Decoder.OpRunning )
   END_RUNG
   RUNG wire#w1
      Contact( "DecoilersHRot".COut.Traslation.InPosition )
      S_Coil( #MB1_Decoder.OpDone )
   END_RUNG
   // the same network as SCL:
   #_w1 := #MB1_Decoder.Code = #"1035_DECOILER_TRANSLATION_MOVE_TO_POS";
   "A01_HMI".MB1.Button.CoilHandling.DecoilersHRot.Translation.MoveToPos := #_w1 AND #MB1_Decoder.OperationPlus;
   IF #_w1 AND ("DecoilersHRot".COut.Traslation.PlusCheckNext OR "DecoilersHRot".COut.Traslation.PlusCheckNext) AND "A01_HMI".MB1.Button.CoilHandling.DecoilersHRot.Translation.MoveToPos THEN
       #MB1_Decoder.OpEnabled := TRUE;
   END_IF;
   IF #_w1 AND NOT "DecoilersHRot".COut.Traslation.Standstill THEN #MB1_Decoder.OpRunning := TRUE; END_IF;
   IF #_w1 AND "DecoilersHRot".COut.Traslation.InPosition THEN #MB1_Decoder.OpDone := TRUE; END_IF;
END_REGION

REGION Network 25: MB1 Code 1041 - Lower Peeler lift up / down
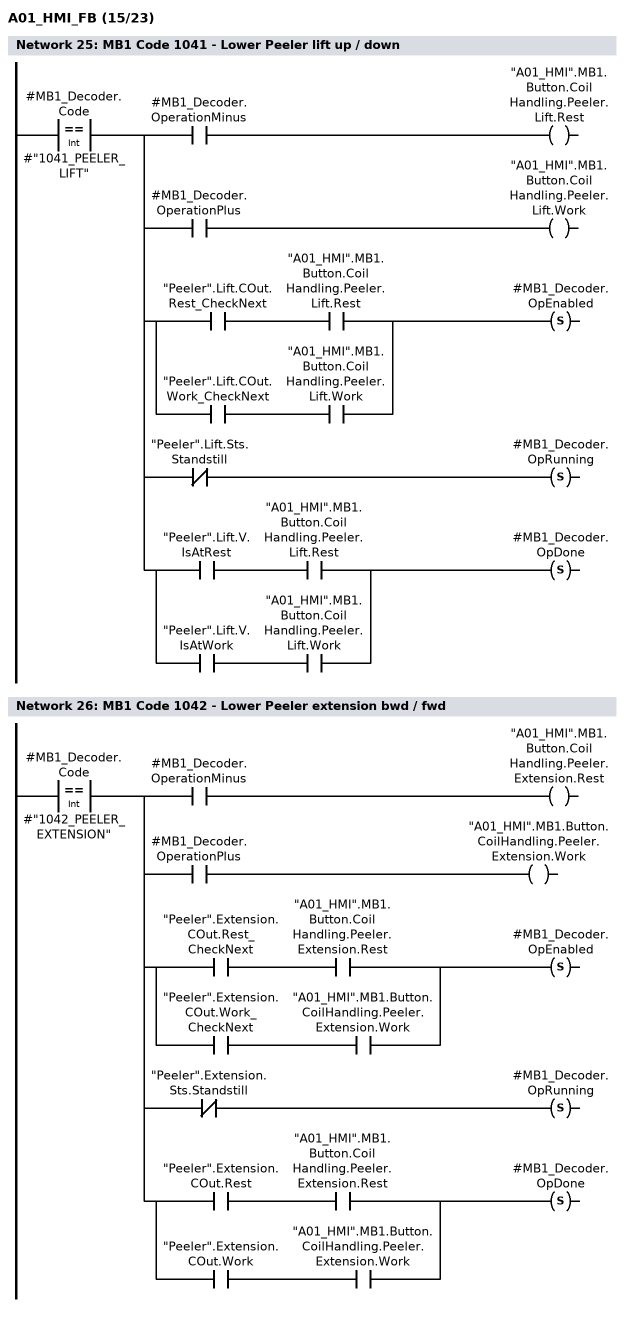
   RUNG wire#powerrail
      { S7_Templates := "SrcType := Int" } EQ_Contact(in1 := #MB1_Decoder.Code, in2 := #"1041_PEELER_LIFT")
      wire#w1
      Contact( #MB1_Decoder.OperationMinus )
      Coil( "A01_HMI".MB1.Button.CoilHandling.Peeler.Lift.Rest )
   END_RUNG
   RUNG wire#w1
      Contact( #MB1_Decoder.OperationPlus )
      Coil( "A01_HMI".MB1.Button.CoilHandling.Peeler.Lift.Work )
   END_RUNG
   RUNG wire#w1
      Contact( "Peeler".Lift.COut.Rest_CheckNext )
      Contact( "A01_HMI".MB1.Button.CoilHandling.Peeler.Lift.Rest )
      wire#w2
      S_Coil( #MB1_Decoder.OpEnabled )
   END_RUNG
   RUNG wire#w1
      Contact( "Peeler".Lift.COut.Work_CheckNext )
      Contact( "A01_HMI".MB1.Button.CoilHandling.Peeler.Lift.Work )
   END_RUNG wire#w2
   RUNG wire#w1
      I_Contact( "Peeler".Lift.Sts.Standstill )
      S_Coil( #MB1_Decoder.OpRunning )
   END_RUNG
   RUNG wire#w1
      Contact( "Peeler".Lift.V.IsAtRest )
      Contact( "A01_HMI".MB1.Button.CoilHandling.Peeler.Lift.Rest )
      wire#w3
      S_Coil( #MB1_Decoder.OpDone )
   END_RUNG
   RUNG wire#w1
      Contact( "Peeler".Lift.V.IsAtWork )
      Contact( "A01_HMI".MB1.Button.CoilHandling.Peeler.Lift.Work )
   END_RUNG wire#w3
   // the same network as SCL:
   #_w1 := #MB1_Decoder.Code = #"1041_PEELER_LIFT";
   "A01_HMI".MB1.Button.CoilHandling.Peeler.Lift.Rest := #_w1 AND #MB1_Decoder.OperationMinus;
   "A01_HMI".MB1.Button.CoilHandling.Peeler.Lift.Work := #_w1 AND #MB1_Decoder.OperationPlus;
   IF #_w1 AND (("Peeler".Lift.COut.Rest_CheckNext AND "A01_HMI".MB1.Button.CoilHandling.Peeler.Lift.Rest) OR ("Peeler".Lift.COut.Work_CheckNext AND "A01_HMI".MB1.Button.CoilHandling.Peeler.Lift.Work)) THEN
       #MB1_Decoder.OpEnabled := TRUE;
   END_IF;
   IF #_w1 AND NOT "Peeler".Lift.Sts.Standstill THEN #MB1_Decoder.OpRunning := TRUE; END_IF;
   IF #_w1 AND (("Peeler".Lift.V.IsAtRest AND "A01_HMI".MB1.Button.CoilHandling.Peeler.Lift.Rest) OR ("Peeler".Lift.V.IsAtWork AND "A01_HMI".MB1.Button.CoilHandling.Peeler.Lift.Work)) THEN
       #MB1_Decoder.OpDone := TRUE;
   END_IF;
END_REGION

REGION Network 26: MB1 Code 1042 - Lower Peeler extension bwd / fwd
   RUNG wire#powerrail
      { S7_Templates := "SrcType := Int" } EQ_Contact(in1 := #MB1_Decoder.Code, in2 := #"1042_PEELER_EXTENSION")
      wire#w1
      Contact( #MB1_Decoder.OperationMinus )
      Coil( "A01_HMI".MB1.Button.CoilHandling.Peeler.Extension.Rest )
   END_RUNG
   RUNG wire#w1
      Contact( #MB1_Decoder.OperationPlus )
      Coil( "A01_HMI".MB1.Button.CoilHandling.Peeler.Extension.Work )
   END_RUNG
   RUNG wire#w1
      Contact( "Peeler".Extension.COut.Rest_CheckNext )
      Contact( "A01_HMI".MB1.Button.CoilHandling.Peeler.Extension.Rest )
      wire#w2
      S_Coil( #MB1_Decoder.OpEnabled )
   END_RUNG
   RUNG wire#w1
      Contact( "Peeler".Extension.COut.Work_CheckNext )
      Contact( "A01_HMI".MB1.Button.CoilHandling.Peeler.Extension.Work )
   END_RUNG wire#w2
   RUNG wire#w1
      I_Contact( "Peeler".Extension.Sts.Standstill )
      S_Coil( #MB1_Decoder.OpRunning )
   END_RUNG
   RUNG wire#w1
      Contact( "Peeler".Extension.COut.Rest )
      Contact( "A01_HMI".MB1.Button.CoilHandling.Peeler.Extension.Rest )
      wire#w3
      S_Coil( #MB1_Decoder.OpDone )
   END_RUNG
   RUNG wire#w1
      Contact( "Peeler".Extension.COut.Work )
      Contact( "A01_HMI".MB1.Button.CoilHandling.Peeler.Extension.Work )
   END_RUNG wire#w3
   // the same network as SCL:
   #_w1 := #MB1_Decoder.Code = #"1042_PEELER_EXTENSION";
   "A01_HMI".MB1.Button.CoilHandling.Peeler.Extension.Rest := #_w1 AND #MB1_Decoder.OperationMinus;
   "A01_HMI".MB1.Button.CoilHandling.Peeler.Extension.Work := #_w1 AND #MB1_Decoder.OperationPlus;
   IF #_w1 AND (("Peeler".Extension.COut.Rest_CheckNext AND "A01_HMI".MB1.Button.CoilHandling.Peeler.Extension.Rest) OR ("Peeler".Extension.COut.Work_CheckNext AND "A01_HMI".MB1.Button.CoilHandling.Peeler.Extension.Work)) THEN
       #MB1_Decoder.OpEnabled := TRUE;
   END_IF;
   IF #_w1 AND NOT "Peeler".Extension.Sts.Standstill THEN #MB1_Decoder.OpRunning := TRUE; END_IF;
   IF #_w1 AND (("Peeler".Extension.COut.Rest AND "A01_HMI".MB1.Button.CoilHandling.Peeler.Extension.Rest) OR ("Peeler".Extension.COut.Work AND "A01_HMI".MB1.Button.CoilHandling.Peeler.Extension.Work)) THEN
       #MB1_Decoder.OpDone := TRUE;
   END_IF;
END_REGION

REGION Network 27: MB1 Code 1051 - Straightener bkw / fwd
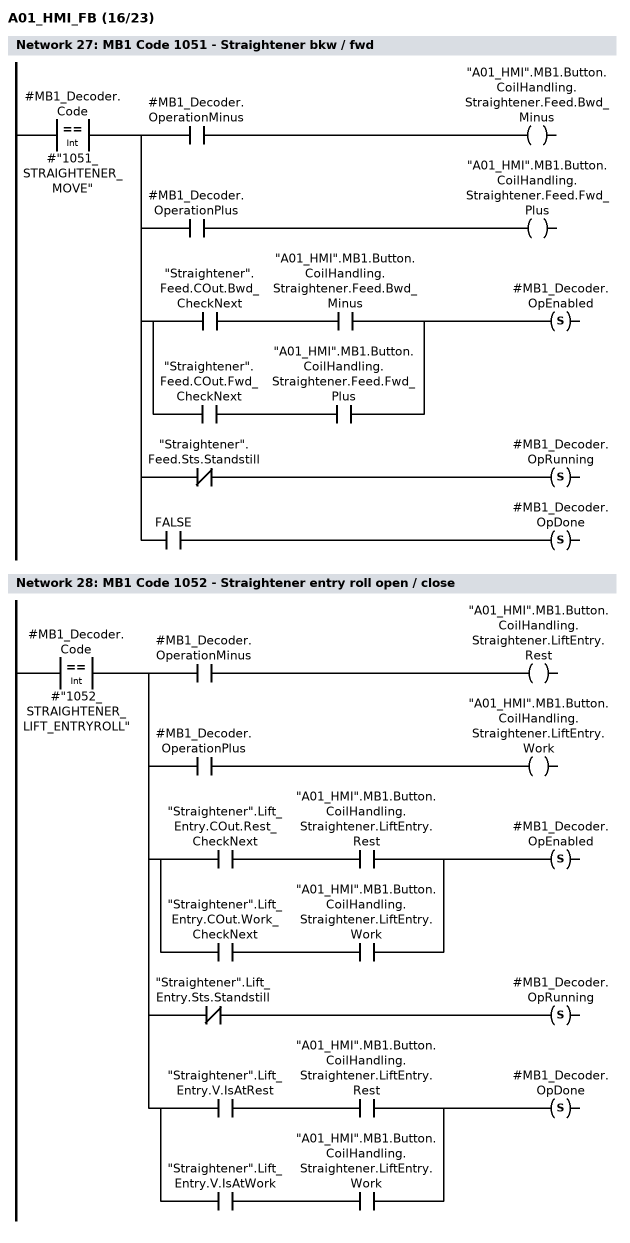
   RUNG wire#powerrail
      { S7_Templates := "SrcType := Int" } EQ_Contact(in1 := #MB1_Decoder.Code, in2 := #"1051_STRAIGHTENER_MOVE")
      wire#w1
      Contact( #MB1_Decoder.OperationMinus )
      Coil( "A01_HMI".MB1.Button.CoilHandling.Straightener.Feed.Bwd_Minus )
   END_RUNG
   RUNG wire#w1
      Contact( #MB1_Decoder.OperationPlus )
      Coil( "A01_HMI".MB1.Button.CoilHandling.Straightener.Feed.Fwd_Plus )
   END_RUNG
   RUNG wire#w1
      Contact( "Straightener".Feed.COut.Bwd_CheckNext )
      Contact( "A01_HMI".MB1.Button.CoilHandling.Straightener.Feed.Bwd_Minus )
      wire#w2
      S_Coil( #MB1_Decoder.OpEnabled )
   END_RUNG
   RUNG wire#w1
      Contact( "Straightener".Feed.COut.Fwd_CheckNext )
      Contact( "A01_HMI".MB1.Button.CoilHandling.Straightener.Feed.Fwd_Plus )
   END_RUNG wire#w2
   RUNG wire#w1
      I_Contact( "Straightener".Feed.Sts.Standstill )
      S_Coil( #MB1_Decoder.OpRunning )
   END_RUNG
   RUNG wire#w1
      Contact( FALSE )
      S_Coil( #MB1_Decoder.OpDone )
   END_RUNG
   // the same network as SCL:
   #_w1 := #MB1_Decoder.Code = #"1051_STRAIGHTENER_MOVE";
   "A01_HMI".MB1.Button.CoilHandling.Straightener.Feed.Bwd_Minus := #_w1 AND #MB1_Decoder.OperationMinus;
   "A01_HMI".MB1.Button.CoilHandling.Straightener.Feed.Fwd_Plus := #_w1 AND #MB1_Decoder.OperationPlus;
   IF #_w1 AND (("Straightener".Feed.COut.Bwd_CheckNext AND "A01_HMI".MB1.Button.CoilHandling.Straightener.Feed.Bwd_Minus) OR ("Straightener".Feed.COut.Fwd_CheckNext AND "A01_HMI".MB1.Button.CoilHandling.Straightener.Feed.Fwd_Plus)) THEN
       #MB1_Decoder.OpEnabled := TRUE;
   END_IF;
   IF #_w1 AND NOT "Straightener".Feed.Sts.Standstill THEN #MB1_Decoder.OpRunning := TRUE; END_IF;
   IF #_w1 AND FALSE THEN #MB1_Decoder.OpDone := TRUE; END_IF;
END_REGION

REGION Network 28: MB1 Code 1052 - Straightener entry roll open / close
   RUNG wire#powerrail
      { S7_Templates := "SrcType := Int" } EQ_Contact(in1 := #MB1_Decoder.Code, in2 := #"1052_STRAIGHTENER_LIFT_ENTRYROLL")
      wire#w1
      Contact( #MB1_Decoder.OperationMinus )
      Coil( "A01_HMI".MB1.Button.CoilHandling.Straightener.LiftEntry.Rest )
   END_RUNG
   RUNG wire#w1
      Contact( #MB1_Decoder.OperationPlus )
      Coil( "A01_HMI".MB1.Button.CoilHandling.Straightener.LiftEntry.Work )
   END_RUNG
   RUNG wire#w1
      Contact( "Straightener".Lift_Entry.COut.Rest_CheckNext )
      Contact( "A01_HMI".MB1.Button.CoilHandling.Straightener.LiftEntry.Rest )
      wire#w2
      S_Coil( #MB1_Decoder.OpEnabled )
   END_RUNG
   RUNG wire#w1
      Contact( "Straightener".Lift_Entry.COut.Work_CheckNext )
      Contact( "A01_HMI".MB1.Button.CoilHandling.Straightener.LiftEntry.Work )
   END_RUNG wire#w2
   RUNG wire#w1
      I_Contact( "Straightener".Lift_Entry.Sts.Standstill )
      S_Coil( #MB1_Decoder.OpRunning )
   END_RUNG
   RUNG wire#w1
      Contact( "Straightener".Lift_Entry.V.IsAtRest )
      Contact( "A01_HMI".MB1.Button.CoilHandling.Straightener.LiftEntry.Rest )
      wire#w3
      S_Coil( #MB1_Decoder.OpDone )
   END_RUNG
   RUNG wire#w1
      Contact( "Straightener".Lift_Entry.V.IsAtWork )
      Contact( "A01_HMI".MB1.Button.CoilHandling.Straightener.LiftEntry.Work )
   END_RUNG wire#w3
   // the same network as SCL:
   #_w1 := #MB1_Decoder.Code = #"1052_STRAIGHTENER_LIFT_ENTRYROLL";
   "A01_HMI".MB1.Button.CoilHandling.Straightener.LiftEntry.Rest := #_w1 AND #MB1_Decoder.OperationMinus;
   "A01_HMI".MB1.Button.CoilHandling.Straightener.LiftEntry.Work := #_w1 AND #MB1_Decoder.OperationPlus;
   IF #_w1 AND (("Straightener".Lift_Entry.COut.Rest_CheckNext AND "A01_HMI".MB1.Button.CoilHandling.Straightener.LiftEntry.Rest) OR ("Straightener".Lift_Entry.COut.Work_CheckNext AND "A01_HMI".MB1.Button.CoilHandling.Straightener.LiftEntry.Work)) THEN
       #MB1_Decoder.OpEnabled := TRUE;
   END_IF;
   IF #_w1 AND NOT "Straightener".Lift_Entry.Sts.Standstill THEN #MB1_Decoder.OpRunning := TRUE; END_IF;
   IF #_w1 AND (("Straightener".Lift_Entry.V.IsAtRest AND "A01_HMI".MB1.Button.CoilHandling.Straightener.LiftEntry.Rest) OR ("Straightener".Lift_Entry.V.IsAtWork AND "A01_HMI".MB1.Button.CoilHandling.Straightener.LiftEntry.Work)) THEN
       #MB1_Decoder.OpDone := TRUE;
   END_IF;
END_REGION

REGION Network 29: MB1 Code 1053 - Straightener exit roll open / close
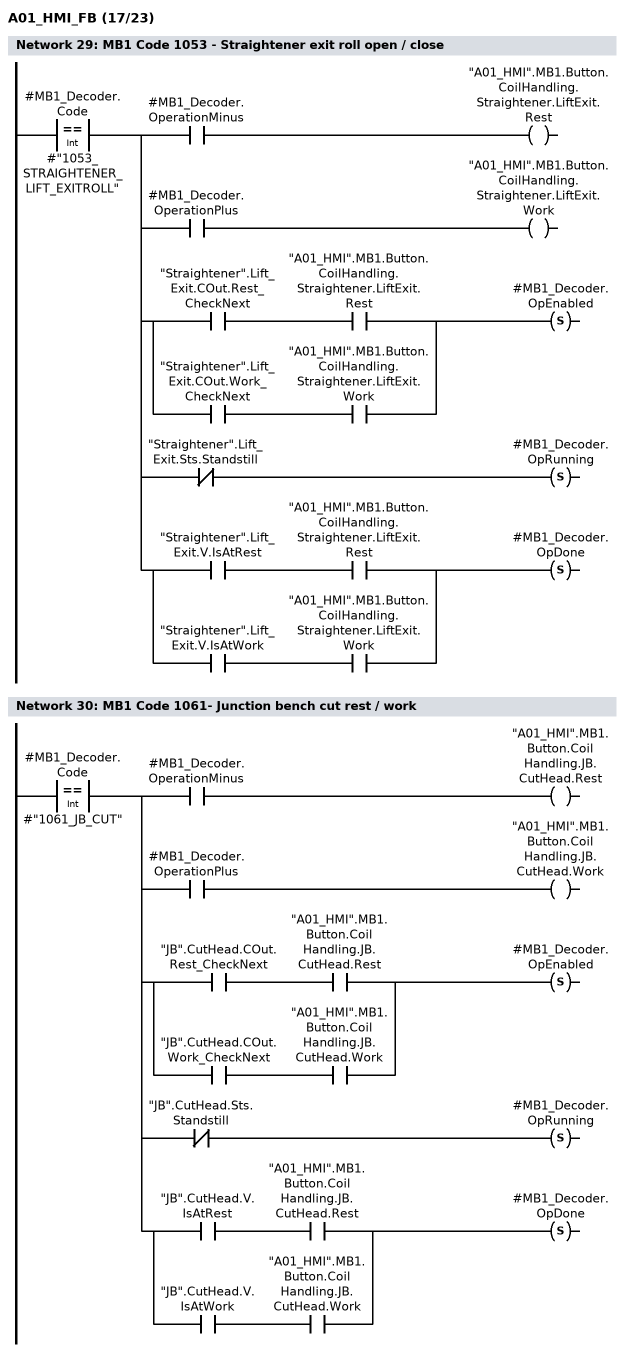
   RUNG wire#powerrail
      { S7_Templates := "SrcType := Int" } EQ_Contact(in1 := #MB1_Decoder.Code, in2 := #"1053_STRAIGHTENER_LIFT_EXITROLL")
      wire#w1
      Contact( #MB1_Decoder.OperationMinus )
      Coil( "A01_HMI".MB1.Button.CoilHandling.Straightener.LiftExit.Rest )
   END_RUNG
   RUNG wire#w1
      Contact( #MB1_Decoder.OperationPlus )
      Coil( "A01_HMI".MB1.Button.CoilHandling.Straightener.LiftExit.Work )
   END_RUNG
   RUNG wire#w1
      Contact( "Straightener".Lift_Exit.COut.Rest_CheckNext )
      Contact( "A01_HMI".MB1.Button.CoilHandling.Straightener.LiftExit.Rest )
      wire#w2
      S_Coil( #MB1_Decoder.OpEnabled )
   END_RUNG
   RUNG wire#w1
      Contact( "Straightener".Lift_Exit.COut.Work_CheckNext )
      Contact( "A01_HMI".MB1.Button.CoilHandling.Straightener.LiftExit.Work )
   END_RUNG wire#w2
   RUNG wire#w1
      I_Contact( "Straightener".Lift_Exit.Sts.Standstill )
      S_Coil( #MB1_Decoder.OpRunning )
   END_RUNG
   RUNG wire#w1
      Contact( "Straightener".Lift_Exit.V.IsAtRest )
      Contact( "A01_HMI".MB1.Button.CoilHandling.Straightener.LiftExit.Rest )
      wire#w3
      S_Coil( #MB1_Decoder.OpDone )
   END_RUNG
   RUNG wire#w1
      Contact( "Straightener".Lift_Exit.V.IsAtWork )
      Contact( "A01_HMI".MB1.Button.CoilHandling.Straightener.LiftExit.Work )
   END_RUNG wire#w3
   // the same network as SCL:
   #_w1 := #MB1_Decoder.Code = #"1053_STRAIGHTENER_LIFT_EXITROLL";
   "A01_HMI".MB1.Button.CoilHandling.Straightener.LiftExit.Rest := #_w1 AND #MB1_Decoder.OperationMinus;
   "A01_HMI".MB1.Button.CoilHandling.Straightener.LiftExit.Work := #_w1 AND #MB1_Decoder.OperationPlus;
   IF #_w1 AND (("Straightener".Lift_Exit.COut.Rest_CheckNext AND "A01_HMI".MB1.Button.CoilHandling.Straightener.LiftExit.Rest) OR ("Straightener".Lift_Exit.COut.Work_CheckNext AND "A01_HMI".MB1.Button.CoilHandling.Straightener.LiftExit.Work)) THEN
       #MB1_Decoder.OpEnabled := TRUE;
   END_IF;
   IF #_w1 AND NOT "Straightener".Lift_Exit.Sts.Standstill THEN #MB1_Decoder.OpRunning := TRUE; END_IF;
   IF #_w1 AND (("Straightener".Lift_Exit.V.IsAtRest AND "A01_HMI".MB1.Button.CoilHandling.Straightener.LiftExit.Rest) OR ("Straightener".Lift_Exit.V.IsAtWork AND "A01_HMI".MB1.Button.CoilHandling.Straightener.LiftExit.Work)) THEN
       #MB1_Decoder.OpDone := TRUE;
   END_IF;
END_REGION

REGION Network 30: MB1 Code 1061- Junction bench cut rest / work
   RUNG wire#powerrail
      { S7_Templates := "SrcType := Int" } EQ_Contact(in1 := #MB1_Decoder.Code, in2 := #"1061_JB_CUT")
      wire#w1
      Contact( #MB1_Decoder.OperationMinus )
      Coil( "A01_HMI".MB1.Button.CoilHandling.JB.CutHead.Rest )
   END_RUNG
   RUNG wire#w1
      Contact( #MB1_Decoder.OperationPlus )
      Coil( "A01_HMI".MB1.Button.CoilHandling.JB.CutHead.Work )
   END_RUNG
   RUNG wire#w1
      Contact( "JB".CutHead.COut.Rest_CheckNext )
      Contact( "A01_HMI".MB1.Button.CoilHandling.JB.CutHead.Rest )
      wire#w2
      S_Coil( #MB1_Decoder.OpEnabled )
   END_RUNG
   RUNG wire#w1
      Contact( "JB".CutHead.COut.Work_CheckNext )
      Contact( "A01_HMI".MB1.Button.CoilHandling.JB.CutHead.Work )
   END_RUNG wire#w2
   RUNG wire#w1
      I_Contact( "JB".CutHead.Sts.Standstill )
      S_Coil( #MB1_Decoder.OpRunning )
   END_RUNG
   RUNG wire#w1
      Contact( "JB".CutHead.V.IsAtRest )
      Contact( "A01_HMI".MB1.Button.CoilHandling.JB.CutHead.Rest )
      wire#w3
      S_Coil( #MB1_Decoder.OpDone )
   END_RUNG
   RUNG wire#w1
      Contact( "JB".CutHead.V.IsAtWork )
      Contact( "A01_HMI".MB1.Button.CoilHandling.JB.CutHead.Work )
   END_RUNG wire#w3
   // the same network as SCL:
   #_w1 := #MB1_Decoder.Code = #"1061_JB_CUT";
   "A01_HMI".MB1.Button.CoilHandling.JB.CutHead.Rest := #_w1 AND #MB1_Decoder.OperationMinus;
   "A01_HMI".MB1.Button.CoilHandling.JB.CutHead.Work := #_w1 AND #MB1_Decoder.OperationPlus;
   IF #_w1 AND (("JB".CutHead.COut.Rest_CheckNext AND "A01_HMI".MB1.Button.CoilHandling.JB.CutHead.Rest) OR ("JB".CutHead.COut.Work_CheckNext AND "A01_HMI".MB1.Button.CoilHandling.JB.CutHead.Work)) THEN
       #MB1_Decoder.OpEnabled := TRUE;
   END_IF;
   IF #_w1 AND NOT "JB".CutHead.Sts.Standstill THEN #MB1_Decoder.OpRunning := TRUE; END_IF;
   IF #_w1 AND (("JB".CutHead.V.IsAtRest AND "A01_HMI".MB1.Button.CoilHandling.JB.CutHead.Rest) OR ("JB".CutHead.V.IsAtWork AND "A01_HMI".MB1.Button.CoilHandling.JB.CutHead.Work)) THEN
       #MB1_Decoder.OpDone := TRUE;
   END_IF;
END_REGION

REGION Network 31: MB1 Code 1062 - Junction bench torch bkw / fwd
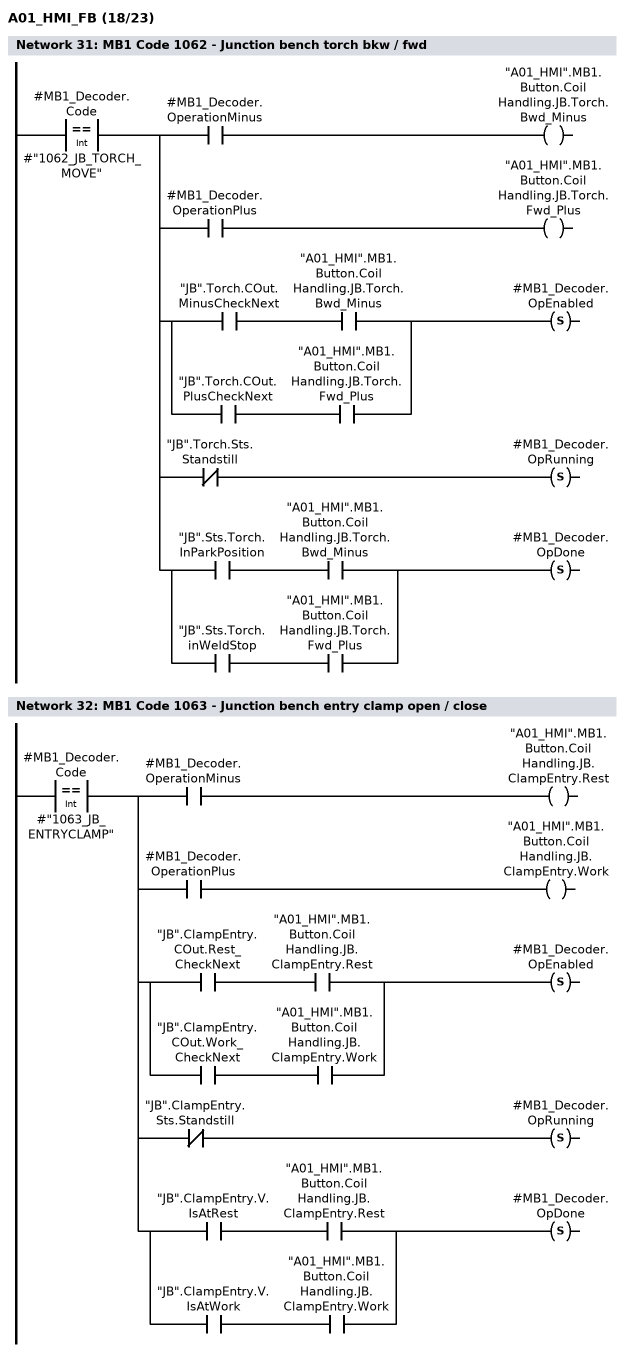
   RUNG wire#powerrail
      { S7_Templates := "SrcType := Int" } EQ_Contact(in1 := #MB1_Decoder.Code, in2 := #"1062_JB_TORCH_MOVE")
      wire#w1
      Contact( #MB1_Decoder.OperationMinus )
      Coil( "A01_HMI".MB1.Button.CoilHandling.JB.Torch.Bwd_Minus )
   END_RUNG
   RUNG wire#w1
      Contact( #MB1_Decoder.OperationPlus )
      Coil( "A01_HMI".MB1.Button.CoilHandling.JB.Torch.Fwd_Plus )
   END_RUNG
   RUNG wire#w1
      Contact( "JB".Torch.COut.MinusCheckNext )
      Contact( "A01_HMI".MB1.Button.CoilHandling.JB.Torch.Bwd_Minus )
      wire#w2
      S_Coil( #MB1_Decoder.OpEnabled )
   END_RUNG
   RUNG wire#w1
      Contact( "JB".Torch.COut.PlusCheckNext )
      Contact( "A01_HMI".MB1.Button.CoilHandling.JB.Torch.Fwd_Plus )
   END_RUNG wire#w2
   RUNG wire#w1
      I_Contact( "JB".Torch.Sts.Standstill )
      S_Coil( #MB1_Decoder.OpRunning )
   END_RUNG
   RUNG wire#w1
      Contact( "JB".Sts.Torch.InParkPosition )
      Contact( "A01_HMI".MB1.Button.CoilHandling.JB.Torch.Bwd_Minus )
      wire#w3
      S_Coil( #MB1_Decoder.OpDone )
   END_RUNG
   RUNG wire#w1
      Contact( "JB".Sts.Torch.inWeldStop )
      Contact( "A01_HMI".MB1.Button.CoilHandling.JB.Torch.Fwd_Plus )
   END_RUNG wire#w3
   // the same network as SCL:
   #_w1 := #MB1_Decoder.Code = #"1062_JB_TORCH_MOVE";
   "A01_HMI".MB1.Button.CoilHandling.JB.Torch.Bwd_Minus := #_w1 AND #MB1_Decoder.OperationMinus;
   "A01_HMI".MB1.Button.CoilHandling.JB.Torch.Fwd_Plus := #_w1 AND #MB1_Decoder.OperationPlus;
   IF #_w1 AND (("JB".Torch.COut.MinusCheckNext AND "A01_HMI".MB1.Button.CoilHandling.JB.Torch.Bwd_Minus) OR ("JB".Torch.COut.PlusCheckNext AND "A01_HMI".MB1.Button.CoilHandling.JB.Torch.Fwd_Plus)) THEN
       #MB1_Decoder.OpEnabled := TRUE;
   END_IF;
   IF #_w1 AND NOT "JB".Torch.Sts.Standstill THEN #MB1_Decoder.OpRunning := TRUE; END_IF;
   IF #_w1 AND (("JB".Sts.Torch.InParkPosition AND "A01_HMI".MB1.Button.CoilHandling.JB.Torch.Bwd_Minus) OR ("JB".Sts.Torch.inWeldStop AND "A01_HMI".MB1.Button.CoilHandling.JB.Torch.Fwd_Plus)) THEN
       #MB1_Decoder.OpDone := TRUE;
   END_IF;
END_REGION

REGION Network 32: MB1 Code 1063 - Junction bench entry clamp open / close
   RUNG wire#powerrail
      { S7_Templates := "SrcType := Int" } EQ_Contact(in1 := #MB1_Decoder.Code, in2 := #"1063_JB_ENTRYCLAMP")
      wire#w1
      Contact( #MB1_Decoder.OperationMinus )
      Coil( "A01_HMI".MB1.Button.CoilHandling.JB.ClampEntry.Rest )
   END_RUNG
   RUNG wire#w1
      Contact( #MB1_Decoder.OperationPlus )
      Coil( "A01_HMI".MB1.Button.CoilHandling.JB.ClampEntry.Work )
   END_RUNG
   RUNG wire#w1
      Contact( "JB".ClampEntry.COut.Rest_CheckNext )
      Contact( "A01_HMI".MB1.Button.CoilHandling.JB.ClampEntry.Rest )
      wire#w2
      S_Coil( #MB1_Decoder.OpEnabled )
   END_RUNG
   RUNG wire#w1
      Contact( "JB".ClampEntry.COut.Work_CheckNext )
      Contact( "A01_HMI".MB1.Button.CoilHandling.JB.ClampEntry.Work )
   END_RUNG wire#w2
   RUNG wire#w1
      I_Contact( "JB".ClampEntry.Sts.Standstill )
      S_Coil( #MB1_Decoder.OpRunning )
   END_RUNG
   RUNG wire#w1
      Contact( "JB".ClampEntry.V.IsAtRest )
      Contact( "A01_HMI".MB1.Button.CoilHandling.JB.ClampEntry.Rest )
      wire#w3
      S_Coil( #MB1_Decoder.OpDone )
   END_RUNG
   RUNG wire#w1
      Contact( "JB".ClampEntry.V.IsAtWork )
      Contact( "A01_HMI".MB1.Button.CoilHandling.JB.ClampEntry.Work )
   END_RUNG wire#w3
   // the same network as SCL:
   #_w1 := #MB1_Decoder.Code = #"1063_JB_ENTRYCLAMP";
   "A01_HMI".MB1.Button.CoilHandling.JB.ClampEntry.Rest := #_w1 AND #MB1_Decoder.OperationMinus;
   "A01_HMI".MB1.Button.CoilHandling.JB.ClampEntry.Work := #_w1 AND #MB1_Decoder.OperationPlus;
   IF #_w1 AND (("JB".ClampEntry.COut.Rest_CheckNext AND "A01_HMI".MB1.Button.CoilHandling.JB.ClampEntry.Rest) OR ("JB".ClampEntry.COut.Work_CheckNext AND "A01_HMI".MB1.Button.CoilHandling.JB.ClampEntry.Work)) THEN
       #MB1_Decoder.OpEnabled := TRUE;
   END_IF;
   IF #_w1 AND NOT "JB".ClampEntry.Sts.Standstill THEN #MB1_Decoder.OpRunning := TRUE; END_IF;
   IF #_w1 AND (("JB".ClampEntry.V.IsAtRest AND "A01_HMI".MB1.Button.CoilHandling.JB.ClampEntry.Rest) OR ("JB".ClampEntry.V.IsAtWork AND "A01_HMI".MB1.Button.CoilHandling.JB.ClampEntry.Work)) THEN
       #MB1_Decoder.OpDone := TRUE;
   END_IF;
END_REGION

REGION Network 33: MB1 Code 1064 - Junction bench exit clamp open / close
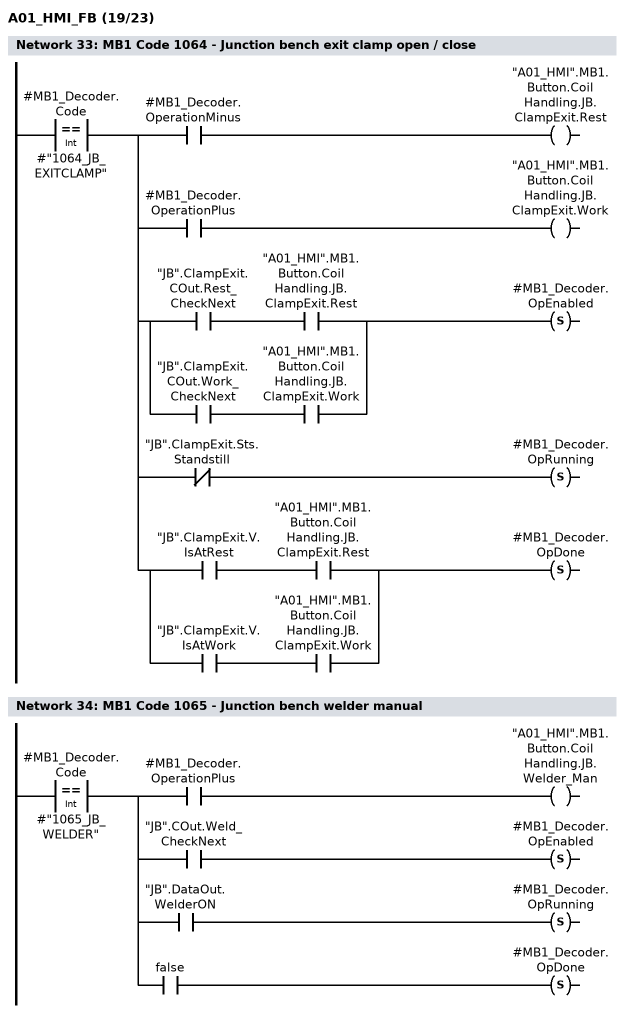
   RUNG wire#powerrail
      { S7_Templates := "SrcType := Int" } EQ_Contact(in1 := #MB1_Decoder.Code, in2 := #"1064_JB_EXITCLAMP")
      wire#w1
      Contact( #MB1_Decoder.OperationMinus )
      Coil( "A01_HMI".MB1.Button.CoilHandling.JB.ClampExit.Rest )
   END_RUNG
   RUNG wire#w1
      Contact( #MB1_Decoder.OperationPlus )
      Coil( "A01_HMI".MB1.Button.CoilHandling.JB.ClampExit.Work )
   END_RUNG
   RUNG wire#w1
      Contact( "JB".ClampExit.COut.Rest_CheckNext )
      Contact( "A01_HMI".MB1.Button.CoilHandling.JB.ClampExit.Rest )
      wire#w2
      S_Coil( #MB1_Decoder.OpEnabled )
   END_RUNG
   RUNG wire#w1
      Contact( "JB".ClampExit.COut.Work_CheckNext )
      Contact( "A01_HMI".MB1.Button.CoilHandling.JB.ClampExit.Work )
   END_RUNG wire#w2
   RUNG wire#w1
      I_Contact( "JB".ClampExit.Sts.Standstill )
      S_Coil( #MB1_Decoder.OpRunning )
   END_RUNG
   RUNG wire#w1
      Contact( "JB".ClampExit.V.IsAtRest )
      Contact( "A01_HMI".MB1.Button.CoilHandling.JB.ClampExit.Rest )
      wire#w3
      S_Coil( #MB1_Decoder.OpDone )
   END_RUNG
   RUNG wire#w1
      Contact( "JB".ClampExit.V.IsAtWork )
      Contact( "A01_HMI".MB1.Button.CoilHandling.JB.ClampExit.Work )
   END_RUNG wire#w3
   // the same network as SCL:
   #_w1 := #MB1_Decoder.Code = #"1064_JB_EXITCLAMP";
   "A01_HMI".MB1.Button.CoilHandling.JB.ClampExit.Rest := #_w1 AND #MB1_Decoder.OperationMinus;
   "A01_HMI".MB1.Button.CoilHandling.JB.ClampExit.Work := #_w1 AND #MB1_Decoder.OperationPlus;
   IF #_w1 AND (("JB".ClampExit.COut.Rest_CheckNext AND "A01_HMI".MB1.Button.CoilHandling.JB.ClampExit.Rest) OR ("JB".ClampExit.COut.Work_CheckNext AND "A01_HMI".MB1.Button.CoilHandling.JB.ClampExit.Work)) THEN
       #MB1_Decoder.OpEnabled := TRUE;
   END_IF;
   IF #_w1 AND NOT "JB".ClampExit.Sts.Standstill THEN #MB1_Decoder.OpRunning := TRUE; END_IF;
   IF #_w1 AND (("JB".ClampExit.V.IsAtRest AND "A01_HMI".MB1.Button.CoilHandling.JB.ClampExit.Rest) OR ("JB".ClampExit.V.IsAtWork AND "A01_HMI".MB1.Button.CoilHandling.JB.ClampExit.Work)) THEN
       #MB1_Decoder.OpDone := TRUE;
   END_IF;
END_REGION

REGION Network 34: MB1 Code 1065 - Junction bench welder manual
   RUNG wire#powerrail
      { S7_Templates := "SrcType := Int" } EQ_Contact(in1 := #MB1_Decoder.Code, in2 := #"1065_JB_WELDER")
      wire#w1
      Contact( #MB1_Decoder.OperationPlus )
      Coil( "A01_HMI".MB1.Button.CoilHandling.JB.Welder_Man )
   END_RUNG
   RUNG wire#w1
      Contact( "JB".COut.Weld_CheckNext )
      S_Coil( #MB1_Decoder.OpEnabled )
   END_RUNG
   RUNG wire#w1
      Contact( "JB".DataOut.WelderON )
      S_Coil( #MB1_Decoder.OpRunning )
   END_RUNG
   RUNG wire#w1
      Contact( false )
      S_Coil( #MB1_Decoder.OpDone )
   END_RUNG
   // the same network as SCL:
   #_w1 := #MB1_Decoder.Code = #"1065_JB_WELDER";
   "A01_HMI".MB1.Button.CoilHandling.JB.Welder_Man := #_w1 AND #MB1_Decoder.OperationPlus;
   IF #_w1 AND "JB".COut.Weld_CheckNext THEN #MB1_Decoder.OpEnabled := TRUE; END_IF;
   IF #_w1 AND "JB".DataOut.WelderON THEN #MB1_Decoder.OpRunning := TRUE; END_IF;
   IF #_w1 AND false THEN #MB1_Decoder.OpDone := TRUE; END_IF;
END_REGION

REGION Network 35: MB1 Code 1066 - Junction bench welding cycle
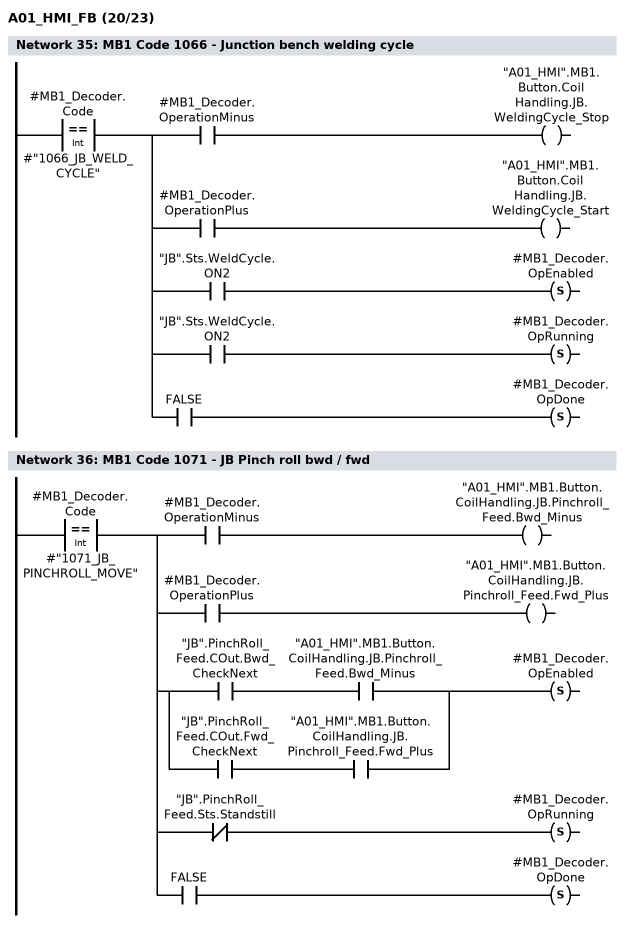
   RUNG wire#powerrail
      { S7_Templates := "SrcType := Int" } EQ_Contact(in1 := #MB1_Decoder.Code, in2 := #"1066_JB_WELD_CYCLE")
      wire#w1
      Contact( #MB1_Decoder.OperationMinus )
      Coil( "A01_HMI".MB1.Button.CoilHandling.JB.WeldingCycle_Stop )
   END_RUNG
   RUNG wire#w1
      Contact( #MB1_Decoder.OperationPlus )
      Coil( "A01_HMI".MB1.Button.CoilHandling.JB.WeldingCycle_Start )
   END_RUNG
   RUNG wire#w1
      Contact( "JB".Sts.WeldCycle.ON2 )
      S_Coil( #MB1_Decoder.OpEnabled )
   END_RUNG
   RUNG wire#w1
      Contact( "JB".Sts.WeldCycle.ON2 )
      S_Coil( #MB1_Decoder.OpRunning )
   END_RUNG
   RUNG wire#w1
      Contact( FALSE )
      S_Coil( #MB1_Decoder.OpDone )
   END_RUNG
   // the same network as SCL:
   #_w1 := #MB1_Decoder.Code = #"1066_JB_WELD_CYCLE";
   "A01_HMI".MB1.Button.CoilHandling.JB.WeldingCycle_Stop := #_w1 AND #MB1_Decoder.OperationMinus;
   "A01_HMI".MB1.Button.CoilHandling.JB.WeldingCycle_Start := #_w1 AND #MB1_Decoder.OperationPlus;
   IF #_w1 AND "JB".Sts.WeldCycle.ON2 THEN
       #MB1_Decoder.OpEnabled := TRUE;
       #MB1_Decoder.OpRunning := TRUE;
   END_IF;
   IF #_w1 AND FALSE THEN #MB1_Decoder.OpDone := TRUE; END_IF;
END_REGION

REGION Network 36: MB1 Code 1071 - JB Pinch roll bwd / fwd
   RUNG wire#powerrail
      { S7_Templates := "SrcType := Int" } EQ_Contact(in1 := #MB1_Decoder.Code, in2 := #"1071_JB_PINCHROLL_MOVE")
      wire#w1
      Contact( #MB1_Decoder.OperationMinus )
      Coil( "A01_HMI".MB1.Button.CoilHandling.JB.Pinchroll_Feed.Bwd_Minus )
   END_RUNG
   RUNG wire#w1
      Contact( #MB1_Decoder.OperationPlus )
      Coil( "A01_HMI".MB1.Button.CoilHandling.JB.Pinchroll_Feed.Fwd_Plus )
   END_RUNG
   RUNG wire#w1
      Contact( "JB".PinchRoll_Feed.COut.Bwd_CheckNext )
      Contact( "A01_HMI".MB1.Button.CoilHandling.JB.Pinchroll_Feed.Bwd_Minus )
      wire#w2
      S_Coil( #MB1_Decoder.OpEnabled )
   END_RUNG
   RUNG wire#w1
      Contact( "JB".PinchRoll_Feed.COut.Fwd_CheckNext )
      Contact( "A01_HMI".MB1.Button.CoilHandling.JB.Pinchroll_Feed.Fwd_Plus )
   END_RUNG wire#w2
   RUNG wire#w1
      I_Contact( "JB".PinchRoll_Feed.Sts.Standstill )
      S_Coil( #MB1_Decoder.OpRunning )
   END_RUNG
   RUNG wire#w1
      Contact( FALSE )
      S_Coil( #MB1_Decoder.OpDone )
   END_RUNG
   // the same network as SCL:
   #_w1 := #MB1_Decoder.Code = #"1071_JB_PINCHROLL_MOVE";
   "A01_HMI".MB1.Button.CoilHandling.JB.Pinchroll_Feed.Bwd_Minus := #_w1 AND #MB1_Decoder.OperationMinus;
   "A01_HMI".MB1.Button.CoilHandling.JB.Pinchroll_Feed.Fwd_Plus := #_w1 AND #MB1_Decoder.OperationPlus;
   IF #_w1 AND (("JB".PinchRoll_Feed.COut.Bwd_CheckNext AND "A01_HMI".MB1.Button.CoilHandling.JB.Pinchroll_Feed.Bwd_Minus) OR ("JB".PinchRoll_Feed.COut.Fwd_CheckNext AND "A01_HMI".MB1.Button.CoilHandling.JB.Pinchroll_Feed.Fwd_Plus)) THEN
       #MB1_Decoder.OpEnabled := TRUE;
   END_IF;
   IF #_w1 AND NOT "JB".PinchRoll_Feed.Sts.Standstill THEN #MB1_Decoder.OpRunning := TRUE; END_IF;
   IF #_w1 AND FALSE THEN #MB1_Decoder.OpDone := TRUE; END_IF;
END_REGION

REGION Network 37: MB1 Code 1072 - JB Pinch roll lift open / close
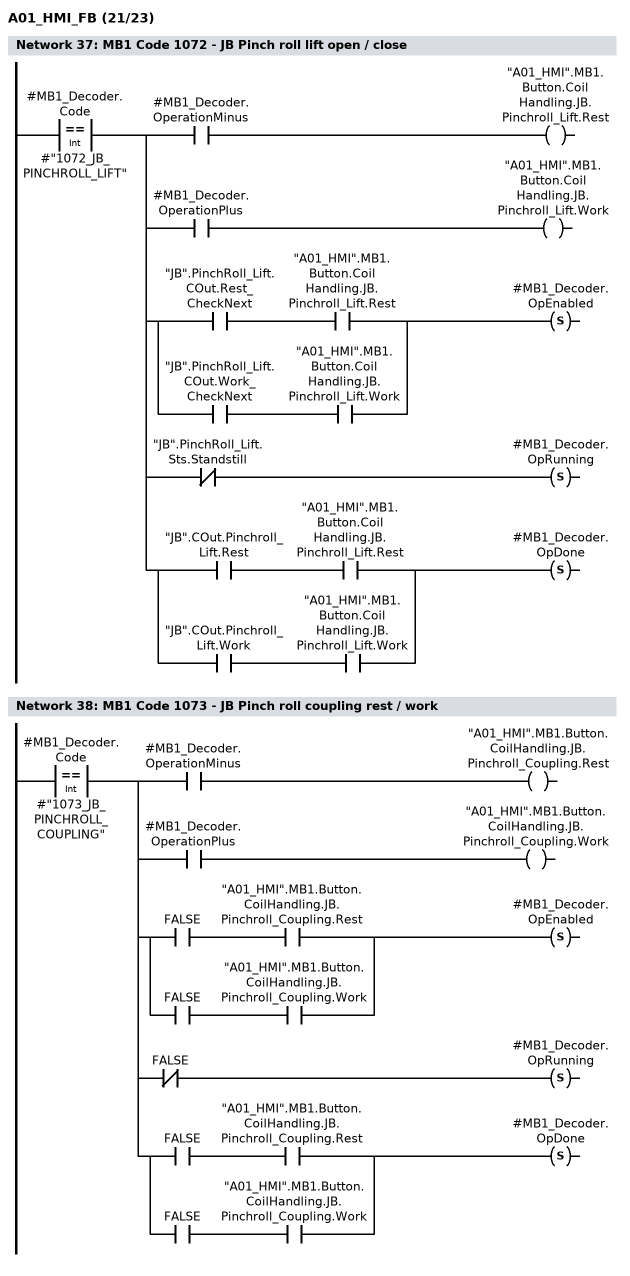
   RUNG wire#powerrail
      { S7_Templates := "SrcType := Int" } EQ_Contact(in1 := #MB1_Decoder.Code, in2 := #"1072_JB_PINCHROLL_LIFT")
      wire#w1
      Contact( #MB1_Decoder.OperationMinus )
      Coil( "A01_HMI".MB1.Button.CoilHandling.JB.Pinchroll_Lift.Rest )
   END_RUNG
   RUNG wire#w1
      Contact( #MB1_Decoder.OperationPlus )
      Coil( "A01_HMI".MB1.Button.CoilHandling.JB.Pinchroll_Lift.Work )
   END_RUNG
   RUNG wire#w1
      Contact( "JB".PinchRoll_Lift.COut.Rest_CheckNext )
      Contact( "A01_HMI".MB1.Button.CoilHandling.JB.Pinchroll_Lift.Rest )
      wire#w2
      S_Coil( #MB1_Decoder.OpEnabled )
   END_RUNG
   RUNG wire#w1
      Contact( "JB".PinchRoll_Lift.COut.Work_CheckNext )
      Contact( "A01_HMI".MB1.Button.CoilHandling.JB.Pinchroll_Lift.Work )
   END_RUNG wire#w2
   RUNG wire#w1
      I_Contact( "JB".PinchRoll_Lift.Sts.Standstill )
      S_Coil( #MB1_Decoder.OpRunning )
   END_RUNG
   RUNG wire#w1
      Contact( "JB".COut.Pinchroll_Lift.Rest )
      Contact( "A01_HMI".MB1.Button.CoilHandling.JB.Pinchroll_Lift.Rest )
      wire#w3
      S_Coil( #MB1_Decoder.OpDone )
   END_RUNG
   RUNG wire#w1
      Contact( "JB".COut.Pinchroll_Lift.Work )
      Contact( "A01_HMI".MB1.Button.CoilHandling.JB.Pinchroll_Lift.Work )
   END_RUNG wire#w3
   // the same network as SCL:
   #_w1 := #MB1_Decoder.Code = #"1072_JB_PINCHROLL_LIFT";
   "A01_HMI".MB1.Button.CoilHandling.JB.Pinchroll_Lift.Rest := #_w1 AND #MB1_Decoder.OperationMinus;
   "A01_HMI".MB1.Button.CoilHandling.JB.Pinchroll_Lift.Work := #_w1 AND #MB1_Decoder.OperationPlus;
   IF #_w1 AND (("JB".PinchRoll_Lift.COut.Rest_CheckNext AND "A01_HMI".MB1.Button.CoilHandling.JB.Pinchroll_Lift.Rest) OR ("JB".PinchRoll_Lift.COut.Work_CheckNext AND "A01_HMI".MB1.Button.CoilHandling.JB.Pinchroll_Lift.Work)) THEN
       #MB1_Decoder.OpEnabled := TRUE;
   END_IF;
   IF #_w1 AND NOT "JB".PinchRoll_Lift.Sts.Standstill THEN #MB1_Decoder.OpRunning := TRUE; END_IF;
   IF #_w1 AND (("JB".COut.Pinchroll_Lift.Rest AND "A01_HMI".MB1.Button.CoilHandling.JB.Pinchroll_Lift.Rest) OR ("JB".COut.Pinchroll_Lift.Work AND "A01_HMI".MB1.Button.CoilHandling.JB.Pinchroll_Lift.Work)) THEN
       #MB1_Decoder.OpDone := TRUE;
   END_IF;
END_REGION

REGION Network 38: MB1 Code 1073 - JB Pinch roll coupling rest / work
   RUNG wire#powerrail
      { S7_Templates := "SrcType := Int" } EQ_Contact(in1 := #MB1_Decoder.Code, in2 := #"1073_JB_PINCHROLL_COUPLING")
      wire#w1
      Contact( #MB1_Decoder.OperationMinus )
      Coil( "A01_HMI".MB1.Button.CoilHandling.JB.Pinchroll_Coupling.Rest )
   END_RUNG
   RUNG wire#w1
      Contact( #MB1_Decoder.OperationPlus )
      Coil( "A01_HMI".MB1.Button.CoilHandling.JB.Pinchroll_Coupling.Work )
   END_RUNG
   RUNG wire#w1
      Contact( FALSE )
      Contact( "A01_HMI".MB1.Button.CoilHandling.JB.Pinchroll_Coupling.Rest )
      wire#w2
      S_Coil( #MB1_Decoder.OpEnabled )
   END_RUNG
   RUNG wire#w1
      Contact( FALSE )
      Contact( "A01_HMI".MB1.Button.CoilHandling.JB.Pinchroll_Coupling.Work )
   END_RUNG wire#w2
   RUNG wire#w1
      I_Contact( FALSE )
      S_Coil( #MB1_Decoder.OpRunning )
   END_RUNG
   RUNG wire#w1
      Contact( FALSE )
      Contact( "A01_HMI".MB1.Button.CoilHandling.JB.Pinchroll_Coupling.Rest )
      wire#w3
      S_Coil( #MB1_Decoder.OpDone )
   END_RUNG
   RUNG wire#w1
      Contact( FALSE )
      Contact( "A01_HMI".MB1.Button.CoilHandling.JB.Pinchroll_Coupling.Work )
   END_RUNG wire#w3
   // the same network as SCL:
   #_w1 := #MB1_Decoder.Code = #"1073_JB_PINCHROLL_COUPLING";
   "A01_HMI".MB1.Button.CoilHandling.JB.Pinchroll_Coupling.Rest := #_w1 AND #MB1_Decoder.OperationMinus;
   "A01_HMI".MB1.Button.CoilHandling.JB.Pinchroll_Coupling.Work := #_w1 AND #MB1_Decoder.OperationPlus;
   IF #_w1 AND ((FALSE AND "A01_HMI".MB1.Button.CoilHandling.JB.Pinchroll_Coupling.Rest) OR (FALSE AND "A01_HMI".MB1.Button.CoilHandling.JB.Pinchroll_Coupling.Work)) THEN
       #MB1_Decoder.OpEnabled := TRUE;
   END_IF;
   IF #_w1 AND NOT FALSE THEN #MB1_Decoder.OpRunning := TRUE; END_IF;
   IF #_w1 AND ((FALSE AND "A01_HMI".MB1.Button.CoilHandling.JB.Pinchroll_Coupling.Rest) OR (FALSE AND "A01_HMI".MB1.Button.CoilHandling.JB.Pinchroll_Coupling.Work)) THEN
       #MB1_Decoder.OpDone := TRUE;
   END_IF;
END_REGION

REGION Network 39: MB1 Code 1081 - Loop 1 Start / Stop
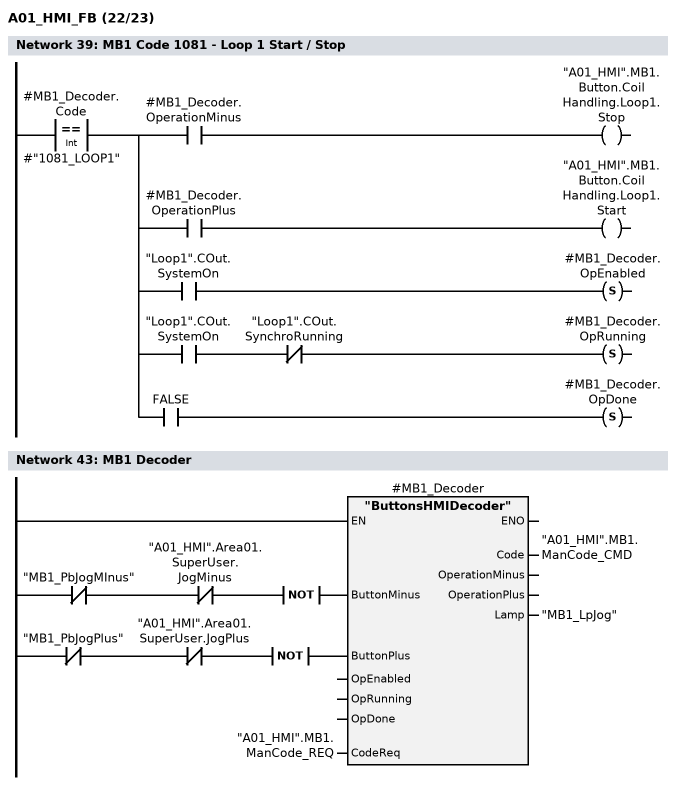
   RUNG wire#powerrail
      { S7_Templates := "SrcType := Int" } EQ_Contact(in1 := #MB1_Decoder.Code, in2 := #"1081_LOOP1")
      wire#w1
      Contact( #MB1_Decoder.OperationMinus )
      Coil( "A01_HMI".MB1.Button.CoilHandling.Loop1.Stop )
   END_RUNG
   RUNG wire#w1
      Contact( #MB1_Decoder.OperationPlus )
      Coil( "A01_HMI".MB1.Button.CoilHandling.Loop1.Start )
   END_RUNG
   RUNG wire#w1
      Contact( "Loop1".COut.SystemOn )
      S_Coil( #MB1_Decoder.OpEnabled )
   END_RUNG
   RUNG wire#w1
      Contact( "Loop1".COut.SystemOn )
      I_Contact( "Loop1".COut.SynchroRunning )
      S_Coil( #MB1_Decoder.OpRunning )
   END_RUNG
   RUNG wire#w1
      Contact( FALSE )
      S_Coil( #MB1_Decoder.OpDone )
   END_RUNG
   // the same network as SCL:
   #_w1 := #MB1_Decoder.Code = #"1081_LOOP1";
   "A01_HMI".MB1.Button.CoilHandling.Loop1.Stop := #_w1 AND #MB1_Decoder.OperationMinus;
   "A01_HMI".MB1.Button.CoilHandling.Loop1.Start := #_w1 AND #MB1_Decoder.OperationPlus;
   IF #_w1 AND "Loop1".COut.SystemOn THEN #MB1_Decoder.OpEnabled := TRUE; END_IF;
   IF #_w1 AND "Loop1".COut.SystemOn AND NOT "Loop1".COut.SynchroRunning THEN
       #MB1_Decoder.OpRunning := TRUE;
   END_IF;
   IF #_w1 AND FALSE THEN #MB1_Decoder.OpDone := TRUE; END_IF;
END_REGION

REGION Network 40: >
END_REGION

REGION Network 41: >
END_REGION

REGION Network 42: >
END_REGION

REGION Network 43: MB1 Decoder
   RUNG wire#powerrail
      #MB1_Decoder(ButtonMinus := wire#w1, ButtonPlus := wire#w2, OpEnabled :=, OpRunning :=, OpDone :=, CodeReq := "A01_HMI".MB1.ManCode_REQ, Code => "A01_HMI".MB1.ManCode_CMD, OperationMinus =>, OperationPlus =>, Lamp => "MB1_LpJog")
   END_RUNG
   RUNG wire#powerrail
      I_Contact( "MB1_PbJogMInus" )
      I_Contact( "A01_HMI".Area01.SuperUser.JogMinus )
      Not()
   END_RUNG wire#w1
   RUNG wire#powerrail
      I_Contact( "MB1_PbJogPlus" )
      I_Contact( "A01_HMI".Area01.SuperUser.JogPlus )
      Not()
   END_RUNG wire#w2
   // the same network as SCL:
   #MB1_Decoder(ButtonMinus := NOT (NOT "MB1_PbJogMInus" AND NOT "A01_HMI".Area01.SuperUser.JogMinus),   // "ButtonsHMIDecoder"
                ButtonPlus := NOT (NOT "MB1_PbJogPlus" AND NOT "A01_HMI".Area01.SuperUser.JogPlus),
                CodeReq := "A01_HMI".MB1.ManCode_REQ,
                Code => "A01_HMI".MB1.ManCode_CMD,
                Lamp => "MB1_LpJog");
END_REGION

REGION Network 44: >
END_REGION

REGION Network 45: >
END_REGION

REGION Network 46: >
END_REGION

REGION Network 47: SINOTTICO
END_REGION

REGION Network 48 (SCL): Decoiler
   "A01_HMI".SYNOPTIC.Decoiler.Decoiler_InLine_DiameterValue := "CoilHandling".COut.Gen.CoilDiameter;
   "A01_HMI".SYNOPTIC.Decoiler.Decoiler_Material_Sts := "CoilHandling".COut.Gen.Material_STS;
   "A01_HMI".SYNOPTIC.Decoiler.Decoiler_InLine_Number := "A01_HMI".SYNOPTIC.Decoiler.Decoiler_InLine_Number;
END_REGION

REGION Network 49: HMI Decoiler in Line
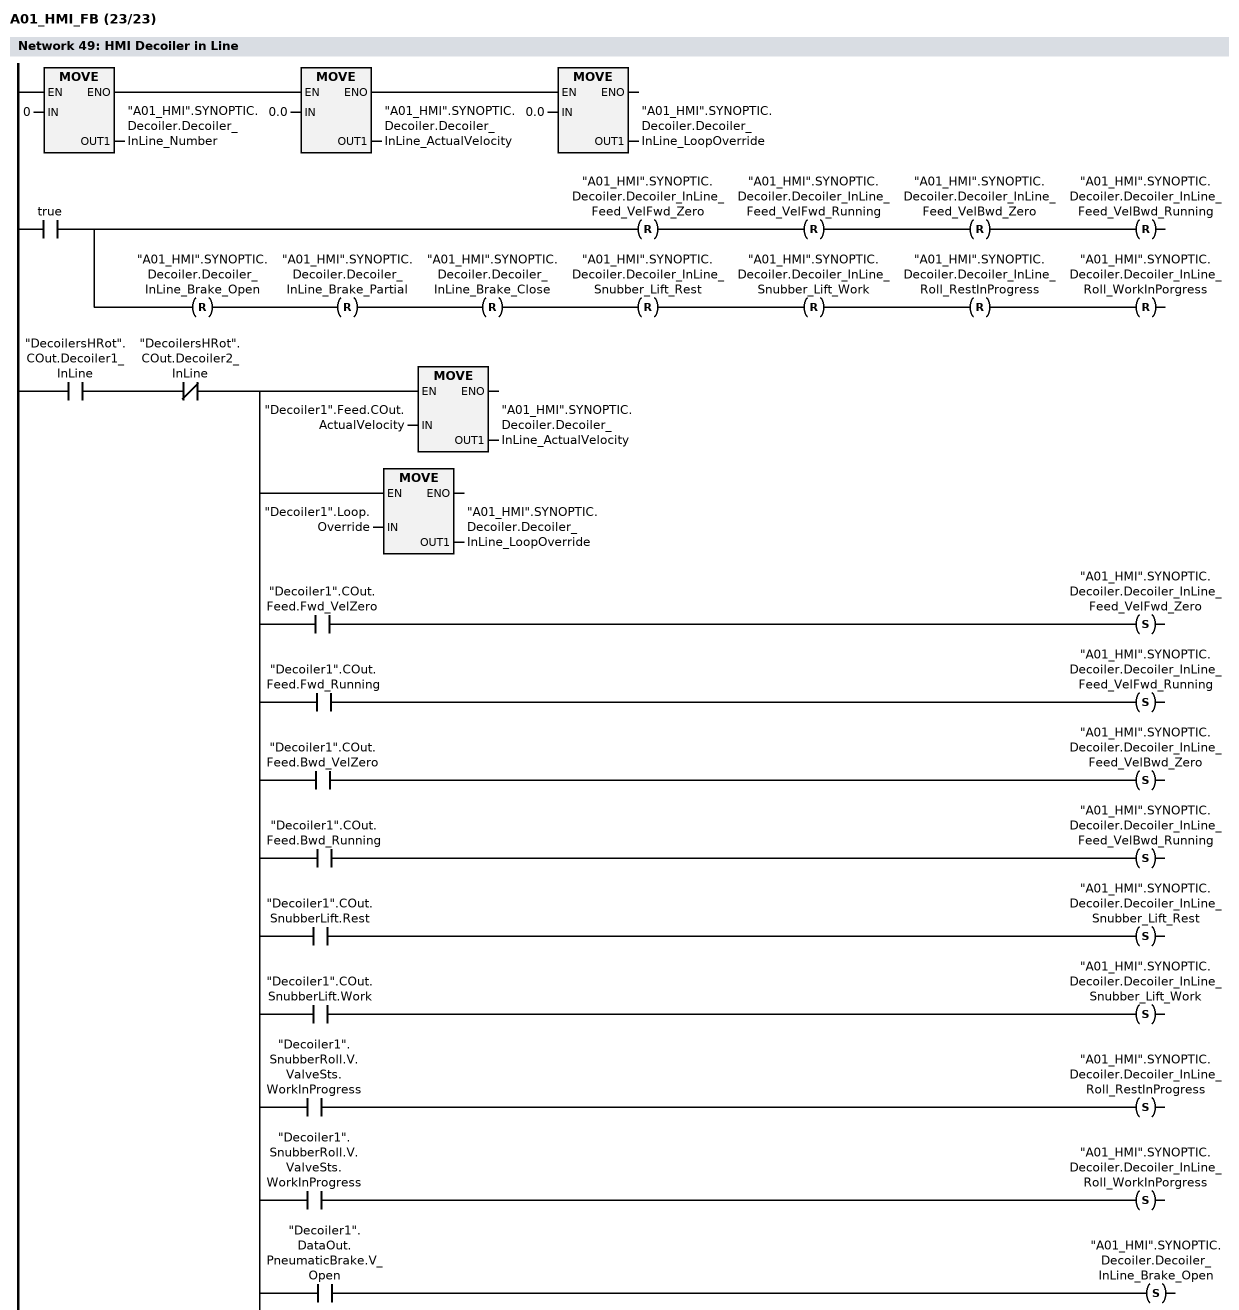
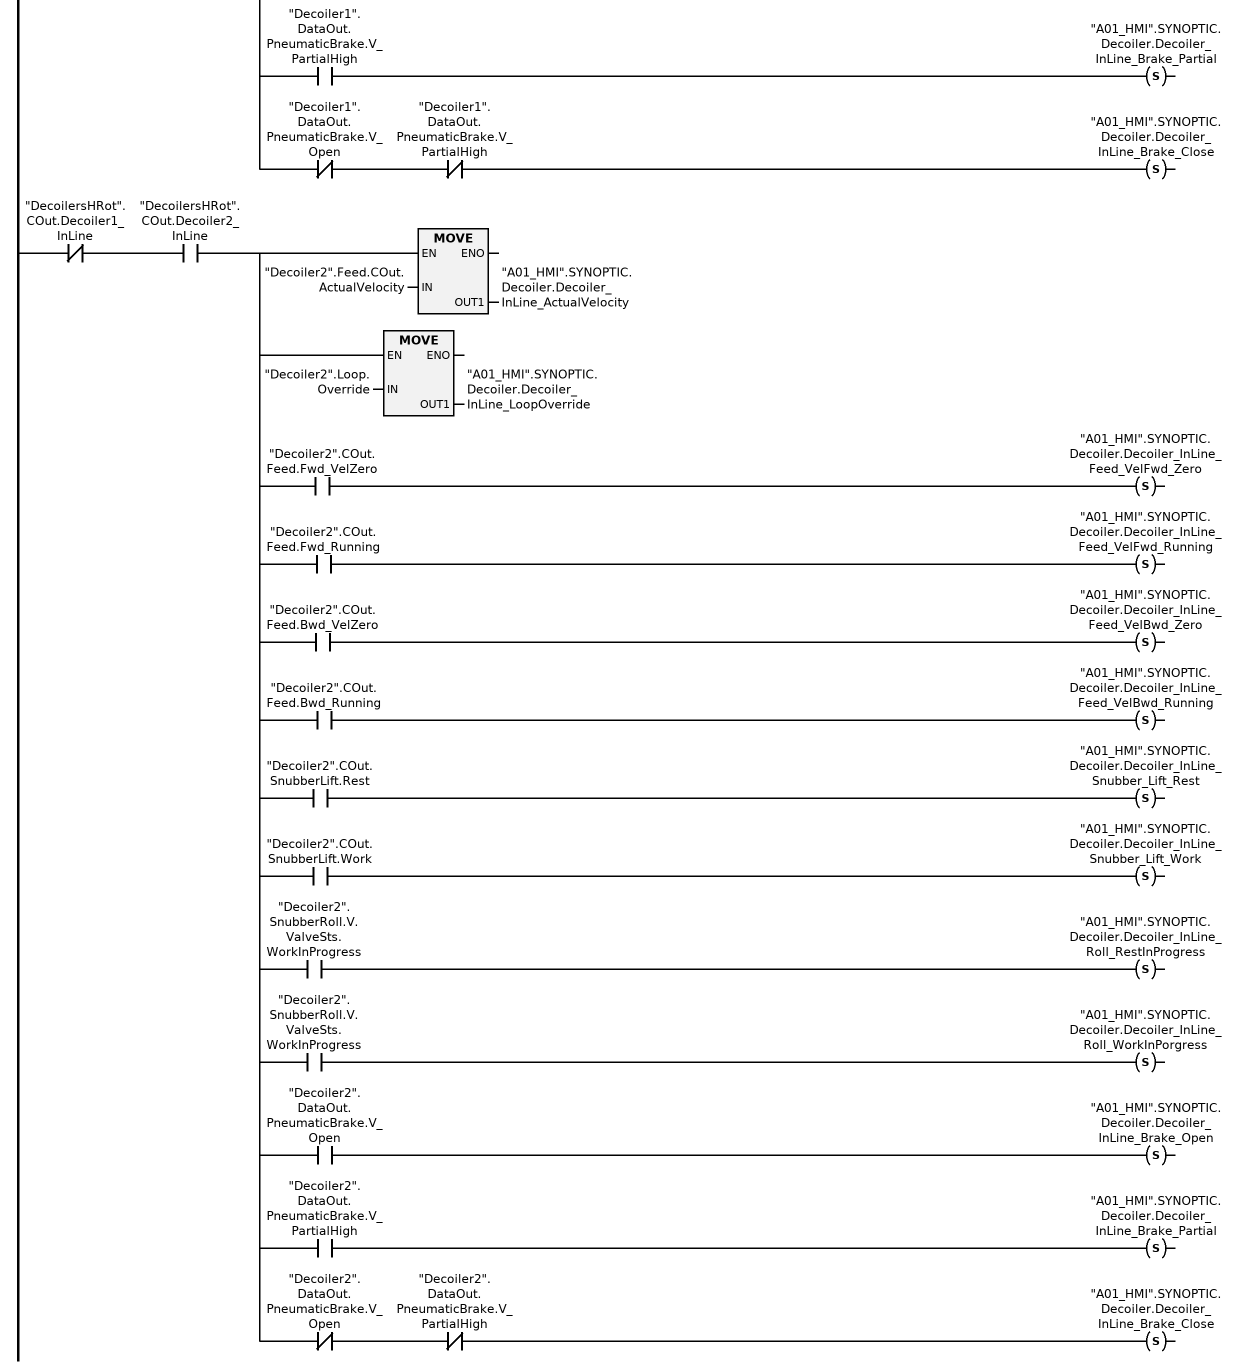
   RUNG wire#powerrail
      { S7_GenerateENO := "TRUE" } Move(in := 0, out1 => "A01_HMI".SYNOPTIC.Decoiler.Decoiler_InLine_Number)
      { S7_GenerateENO := "TRUE" } Move(in := 0.0, out1 => "A01_HMI".SYNOPTIC.Decoiler.Decoiler_InLine_ActualVelocity)
      { S7_GenerateENO := "TRUE" } Move(in := 0.0, out1 => "A01_HMI".SYNOPTIC.Decoiler.Decoiler_InLine_LoopOverride)
   END_RUNG
   RUNG wire#powerrail
      Contact( true )
      wire#w1
      R_Coil( "A01_HMI".SYNOPTIC.Decoiler.Decoiler_InLine_Feed_VelFwd_Zero )
      R_Coil( "A01_HMI".SYNOPTIC.Decoiler.Decoiler_InLine_Feed_VelFwd_Running )
      R_Coil( "A01_HMI".SYNOPTIC.Decoiler.Decoiler_InLine_Feed_VelBwd_Zero )
      R_Coil( "A01_HMI".SYNOPTIC.Decoiler.Decoiler_InLine_Feed_VelBwd_Running )
   END_RUNG
   RUNG wire#w1
      R_Coil( "A01_HMI".SYNOPTIC.Decoiler.Decoiler_InLine_Brake_Open )
      R_Coil( "A01_HMI".SYNOPTIC.Decoiler.Decoiler_InLine_Brake_Partial )
      R_Coil( "A01_HMI".SYNOPTIC.Decoiler.Decoiler_InLine_Brake_Close )
      R_Coil( "A01_HMI".SYNOPTIC.Decoiler.Decoiler_InLine_Snubber_Lift_Rest )
      R_Coil( "A01_HMI".SYNOPTIC.Decoiler.Decoiler_InLine_Snubber_Lift_Work )
      R_Coil( "A01_HMI".SYNOPTIC.Decoiler.Decoiler_InLine_Roll_RestInProgress )
      R_Coil( "A01_HMI".SYNOPTIC.Decoiler.Decoiler_InLine_Roll_WorkInPorgress )
   END_RUNG
   RUNG wire#powerrail
      Contact( "DecoilersHRot".COut.Decoiler1_InLine )
      I_Contact( "DecoilersHRot".COut.Decoiler2_InLine )
      wire#w2
      { S7_GenerateENO := "TRUE" } Move(in := "Decoiler1".Feed.COut.ActualVelocity, out1 => "A01_HMI".SYNOPTIC.Decoiler.Decoiler_InLine_ActualVelocity)
   END_RUNG
   RUNG wire#w2
      { S7_GenerateENO := "TRUE" } Move(in := "Decoiler1".Loop.Override, out1 => "A01_HMI".SYNOPTIC.Decoiler.Decoiler_InLine_LoopOverride)
   END_RUNG
   RUNG wire#w2
      Contact( "Decoiler1".COut.Feed.Fwd_VelZero )
      S_Coil( "A01_HMI".SYNOPTIC.Decoiler.Decoiler_InLine_Feed_VelFwd_Zero )
   END_RUNG
   RUNG wire#w2
      Contact( "Decoiler1".COut.Feed.Fwd_Running )
      S_Coil( "A01_HMI".SYNOPTIC.Decoiler.Decoiler_InLine_Feed_VelFwd_Running )
   END_RUNG
   RUNG wire#w2
      Contact( "Decoiler1".COut.Feed.Bwd_VelZero )
      S_Coil( "A01_HMI".SYNOPTIC.Decoiler.Decoiler_InLine_Feed_VelBwd_Zero )
   END_RUNG
   RUNG wire#w2
      Contact( "Decoiler1".COut.Feed.Bwd_Running )
      S_Coil( "A01_HMI".SYNOPTIC.Decoiler.Decoiler_InLine_Feed_VelBwd_Running )
   END_RUNG
   RUNG wire#w2
      Contact( "Decoiler1".COut.SnubberLift.Rest )
      S_Coil( "A01_HMI".SYNOPTIC.Decoiler.Decoiler_InLine_Snubber_Lift_Rest )
   END_RUNG
   RUNG wire#w2
      Contact( "Decoiler1".COut.SnubberLift.Work )
      S_Coil( "A01_HMI".SYNOPTIC.Decoiler.Decoiler_InLine_Snubber_Lift_Work )
   END_RUNG
   RUNG wire#w2
      Contact( "Decoiler1".SnubberRoll.V.ValveSts.WorkInProgress )
      S_Coil( "A01_HMI".SYNOPTIC.Decoiler.Decoiler_InLine_Roll_RestInProgress )
   END_RUNG
   RUNG wire#w2
      Contact( "Decoiler1".SnubberRoll.V.ValveSts.WorkInProgress )
      S_Coil( "A01_HMI".SYNOPTIC.Decoiler.Decoiler_InLine_Roll_WorkInPorgress )
   END_RUNG
   RUNG wire#w2
      Contact( "Decoiler1".DataOut.PneumaticBrake.V_Open )
      S_Coil( "A01_HMI".SYNOPTIC.Decoiler.Decoiler_InLine_Brake_Open )
   END_RUNG
   RUNG wire#w2
      Contact( "Decoiler1".DataOut.PneumaticBrake.V_PartialHigh )
      S_Coil( "A01_HMI".SYNOPTIC.Decoiler.Decoiler_InLine_Brake_Partial )
   END_RUNG
   RUNG wire#w2
      I_Contact( "Decoiler1".DataOut.PneumaticBrake.V_Open )
      I_Contact( "Decoiler1".DataOut.PneumaticBrake.V_PartialHigh )
      S_Coil( "A01_HMI".SYNOPTIC.Decoiler.Decoiler_InLine_Brake_Close )
   END_RUNG
   RUNG wire#powerrail
      I_Contact( "DecoilersHRot".COut.Decoiler1_InLine )
      Contact( "DecoilersHRot".COut.Decoiler2_InLine )
      wire#w3
      { S7_GenerateENO := "TRUE" } Move(in := "Decoiler2".Feed.COut.ActualVelocity, out1 => "A01_HMI".SYNOPTIC.Decoiler.Decoiler_InLine_ActualVelocity)
   END_RUNG
   RUNG wire#w3
      { S7_GenerateENO := "TRUE" } Move(in := "Decoiler2".Loop.Override, out1 => "A01_HMI".SYNOPTIC.Decoiler.Decoiler_InLine_LoopOverride)
   END_RUNG
   RUNG wire#w3
      Contact( "Decoiler2".COut.Feed.Fwd_VelZero )
      S_Coil( "A01_HMI".SYNOPTIC.Decoiler.Decoiler_InLine_Feed_VelFwd_Zero )
   END_RUNG
   RUNG wire#w3
      Contact( "Decoiler2".COut.Feed.Fwd_Running )
      S_Coil( "A01_HMI".SYNOPTIC.Decoiler.Decoiler_InLine_Feed_VelFwd_Running )
   END_RUNG
   RUNG wire#w3
      Contact( "Decoiler2".COut.Feed.Bwd_VelZero )
      S_Coil( "A01_HMI".SYNOPTIC.Decoiler.Decoiler_InLine_Feed_VelBwd_Zero )
   END_RUNG
   RUNG wire#w3
      Contact( "Decoiler2".COut.Feed.Bwd_Running )
      S_Coil( "A01_HMI".SYNOPTIC.Decoiler.Decoiler_InLine_Feed_VelBwd_Running )
   END_RUNG
   RUNG wire#w3
      Contact( "Decoiler2".COut.SnubberLift.Rest )
      S_Coil( "A01_HMI".SYNOPTIC.Decoiler.Decoiler_InLine_Snubber_Lift_Rest )
   END_RUNG
   RUNG wire#w3
      Contact( "Decoiler2".COut.SnubberLift.Work )
      S_Coil( "A01_HMI".SYNOPTIC.Decoiler.Decoiler_InLine_Snubber_Lift_Work )
   END_RUNG
   RUNG wire#w3
      Contact( "Decoiler2".SnubberRoll.V.ValveSts.WorkInProgress )
      S_Coil( "A01_HMI".SYNOPTIC.Decoiler.Decoiler_InLine_Roll_RestInProgress )
   END_RUNG
   RUNG wire#w3
      Contact( "Decoiler2".SnubberRoll.V.ValveSts.WorkInProgress )
      S_Coil( "A01_HMI".SYNOPTIC.Decoiler.Decoiler_InLine_Roll_WorkInPorgress )
   END_RUNG
   RUNG wire#w3
      Contact( "Decoiler2".DataOut.PneumaticBrake.V_Open )
      S_Coil( "A01_HMI".SYNOPTIC.Decoiler.Decoiler_InLine_Brake_Open )
   END_RUNG
   RUNG wire#w3
      Contact( "Decoiler2".DataOut.PneumaticBrake.V_PartialHigh )
      S_Coil( "A01_HMI".SYNOPTIC.Decoiler.Decoiler_InLine_Brake_Partial )
   END_RUNG
   RUNG wire#w3
      I_Contact( "Decoiler2".DataOut.PneumaticBrake.V_Open )
      I_Contact( "Decoiler2".DataOut.PneumaticBrake.V_PartialHigh )
      S_Coil( "A01_HMI".SYNOPTIC.Decoiler.Decoiler_InLine_Brake_Close )
   END_RUNG
   // the same network as SCL:
   // ENO of a box is taken as its EN; it also drops when the box reports an error
   "A01_HMI".SYNOPTIC.Decoiler.Decoiler_InLine_Number := 0;
   "A01_HMI".SYNOPTIC.Decoiler.Decoiler_InLine_ActualVelocity := 0.0;
   "A01_HMI".SYNOPTIC.Decoiler.Decoiler_InLine_LoopOverride := 0.0;
   IF true THEN
       "A01_HMI".SYNOPTIC.Decoiler.Decoiler_InLine_Feed_VelFwd_Zero := FALSE;
       "A01_HMI".SYNOPTIC.Decoiler.Decoiler_InLine_Feed_VelFwd_Running := FALSE;
       "A01_HMI".SYNOPTIC.Decoiler.Decoiler_InLine_Feed_VelBwd_Zero := FALSE;
       "A01_HMI".SYNOPTIC.Decoiler.Decoiler_InLine_Feed_VelBwd_Running := FALSE;
       "A01_HMI".SYNOPTIC.Decoiler.Decoiler_InLine_Brake_Open := FALSE;
       "A01_HMI".SYNOPTIC.Decoiler.Decoiler_InLine_Brake_Partial := FALSE;
       "A01_HMI".SYNOPTIC.Decoiler.Decoiler_InLine_Brake_Close := FALSE;
       "A01_HMI".SYNOPTIC.Decoiler.Decoiler_InLine_Snubber_Lift_Rest := FALSE;
       "A01_HMI".SYNOPTIC.Decoiler.Decoiler_InLine_Snubber_Lift_Work := FALSE;
       "A01_HMI".SYNOPTIC.Decoiler.Decoiler_InLine_Roll_RestInProgress := FALSE;
       "A01_HMI".SYNOPTIC.Decoiler.Decoiler_InLine_Roll_WorkInPorgress := FALSE;
   END_IF;
   #_w1 := "DecoilersHRot".COut.Decoiler1_InLine AND NOT "DecoilersHRot".COut.Decoiler2_InLine;
   IF #_w1 THEN
       "A01_HMI".SYNOPTIC.Decoiler.Decoiler_InLine_ActualVelocity := "Decoiler1".Feed.COut.ActualVelocity;
       "A01_HMI".SYNOPTIC.Decoiler.Decoiler_InLine_LoopOverride := "Decoiler1".Loop.Override;
   END_IF;
   IF #_w1 AND "Decoiler1".COut.Feed.Fwd_VelZero THEN
       "A01_HMI".SYNOPTIC.Decoiler.Decoiler_InLine_Feed_VelFwd_Zero := TRUE;
   END_IF;
   IF #_w1 AND "Decoiler1".COut.Feed.Fwd_Running THEN
       "A01_HMI".SYNOPTIC.Decoiler.Decoiler_InLine_Feed_VelFwd_Running := TRUE;
   END_IF;
   IF #_w1 AND "Decoiler1".COut.Feed.Bwd_VelZero THEN
       "A01_HMI".SYNOPTIC.Decoiler.Decoiler_InLine_Feed_VelBwd_Zero := TRUE;
   END_IF;
   IF #_w1 AND "Decoiler1".COut.Feed.Bwd_Running THEN
       "A01_HMI".SYNOPTIC.Decoiler.Decoiler_InLine_Feed_VelBwd_Running := TRUE;
   END_IF;
   IF #_w1 AND "Decoiler1".COut.SnubberLift.Rest THEN
       "A01_HMI".SYNOPTIC.Decoiler.Decoiler_InLine_Snubber_Lift_Rest := TRUE;
   END_IF;
   IF #_w1 AND "Decoiler1".COut.SnubberLift.Work THEN
       "A01_HMI".SYNOPTIC.Decoiler.Decoiler_InLine_Snubber_Lift_Work := TRUE;
   END_IF;
   IF #_w1 AND "Decoiler1".SnubberRoll.V.ValveSts.WorkInProgress THEN
       "A01_HMI".SYNOPTIC.Decoiler.Decoiler_InLine_Roll_RestInProgress := TRUE;
       "A01_HMI".SYNOPTIC.Decoiler.Decoiler_InLine_Roll_WorkInPorgress := TRUE;
   END_IF;
   IF #_w1 AND "Decoiler1".DataOut.PneumaticBrake.V_Open THEN
       "A01_HMI".SYNOPTIC.Decoiler.Decoiler_InLine_Brake_Open := TRUE;
   END_IF;
   IF #_w1 AND "Decoiler1".DataOut.PneumaticBrake.V_PartialHigh THEN
       "A01_HMI".SYNOPTIC.Decoiler.Decoiler_InLine_Brake_Partial := TRUE;
   END_IF;
   IF #_w1 AND NOT "Decoiler1".DataOut.PneumaticBrake.V_Open AND NOT "Decoiler1".DataOut.PneumaticBrake.V_PartialHigh THEN
       "A01_HMI".SYNOPTIC.Decoiler.Decoiler_InLine_Brake_Close := TRUE;
   END_IF;
   #_w2 := NOT "DecoilersHRot".COut.Decoiler1_InLine AND "DecoilersHRot".COut.Decoiler2_InLine;
   IF #_w2 THEN
       "A01_HMI".SYNOPTIC.Decoiler.Decoiler_InLine_ActualVelocity := "Decoiler2".Feed.COut.ActualVelocity;
       "A01_HMI".SYNOPTIC.Decoiler.Decoiler_InLine_LoopOverride := "Decoiler2".Loop.Override;
   END_IF;
   IF #_w2 AND "Decoiler2".COut.Feed.Fwd_VelZero THEN
       "A01_HMI".SYNOPTIC.Decoiler.Decoiler_InLine_Feed_VelFwd_Zero := TRUE;
   END_IF;
   IF #_w2 AND "Decoiler2".COut.Feed.Fwd_Running THEN
       "A01_HMI".SYNOPTIC.Decoiler.Decoiler_InLine_Feed_VelFwd_Running := TRUE;
   END_IF;
   IF #_w2 AND "Decoiler2".COut.Feed.Bwd_VelZero THEN
       "A01_HMI".SYNOPTIC.Decoiler.Decoiler_InLine_Feed_VelBwd_Zero := TRUE;
   END_IF;
   IF #_w2 AND "Decoiler2".COut.Feed.Bwd_Running THEN
       "A01_HMI".SYNOPTIC.Decoiler.Decoiler_InLine_Feed_VelBwd_Running := TRUE;
   END_IF;
   IF #_w2 AND "Decoiler2".COut.SnubberLift.Rest THEN
       "A01_HMI".SYNOPTIC.Decoiler.Decoiler_InLine_Snubber_Lift_Rest := TRUE;
   END_IF;
   IF #_w2 AND "Decoiler2".COut.SnubberLift.Work THEN
       "A01_HMI".SYNOPTIC.Decoiler.Decoiler_InLine_Snubber_Lift_Work := TRUE;
   END_IF;
   IF #_w2 AND "Decoiler2".SnubberRoll.V.ValveSts.WorkInProgress THEN
       "A01_HMI".SYNOPTIC.Decoiler.Decoiler_InLine_Roll_RestInProgress := TRUE;
       "A01_HMI".SYNOPTIC.Decoiler.Decoiler_InLine_Roll_WorkInPorgress := TRUE;
   END_IF;
   IF #_w2 AND "Decoiler2".DataOut.PneumaticBrake.V_Open THEN
       "A01_HMI".SYNOPTIC.Decoiler.Decoiler_InLine_Brake_Open := TRUE;
   END_IF;
   IF #_w2 AND "Decoiler2".DataOut.PneumaticBrake.V_PartialHigh THEN
       "A01_HMI".SYNOPTIC.Decoiler.Decoiler_InLine_Brake_Partial := TRUE;
   END_IF;
   IF #_w2 AND NOT "Decoiler2".DataOut.PneumaticBrake.V_Open AND NOT "Decoiler2".DataOut.PneumaticBrake.V_PartialHigh THEN
       "A01_HMI".SYNOPTIC.Decoiler.Decoiler_InLine_Brake_Close := TRUE;
   END_IF;
END_REGION

REGION Network 50 (SCL): Straightner
   "A01_HMI".SYNOPTIC.Straightner.Straight_MatPresence_Entry := "CoilHandling".DataIn.SensorMatPresence_StraightEntry;
   "A01_HMI".SYNOPTIC.Straightner.Straight_MatPresence_Exit := "CoilHandling".DataIn.SensorMatPresence_StraightExit;
   "A01_HMI".SYNOPTIC.Straightner.Straight_ActualVelocity := "Straightener".COut.Feed.ActualVelocity;
END_REGION

REGION Network 51 (SCL): Loop
   "A01_HMI".SYNOPTIC.Loop.Loop_Phc_MinHigh := "Loop1_LsMinHigh";
   "A01_HMI".SYNOPTIC.Loop.Loop_Phc_MaxLow := "Loop1_LsMaxLow";
   "A01_HMI".SYNOPTIC.Loop.Loop_SystemOn := "Loop1".COut.SystemOn;
   "A01_HMI".SYNOPTIC.Loop.Loop_MaterialCounterValid := "Loop1".COut.LoopMaterialCounterValid;
   "A01_HMI".SYNOPTIC.Loop.Loop_MaterialCounter := "Loop1".COut.LoopMaterialCounter;
   "A01_HMI".SYNOPTIC.Loop.Loop_AllowableFeedFwd := "Loop1".COut.Exit_MaxAllowableFeedFwd;
   "A01_HMI".SYNOPTIC.Loop.Loop_ActVelOverrideEntry_Code :="Loop1".COut.Entry_ActVelocityOverride;
   "A01_HMI".SYNOPTIC.Loop.Loop_ActVelOverrideExit_Code :="Loop1".COut.Exit_ActVelocityOverride;
   "A01_HMI".SYNOPTIC.Loop.Loop_MatMissToSynch :="Loop1".COut.LoopMaterialMissingToSynch;
   "A01_HMI".SYNOPTIC.Loop.Loop_MatMissToMaxLow :="Loop1".COut.LoopMaterialMissingToMaxLow;
   "A01_HMI".SYNOPTIC.Loop.Loop_MatMissToMinHigh :="Loop1".COut.LoopMaterialMissingToMinHigh;
   "A01_HMI".SYNOPTIC.Loop.Loop_ActVelOverrideEntry :="Loop1".COut.Entry_VelocityOverride;
   "A01_HMI".SYNOPTIC.Loop.Loop_ActVelOverrideExit :="Loop1".COut.Exit_VelocityOverride;
END_REGION
END_FUNCTION_BLOCK
